LIN {X 0,Y 197.249,Z 148.851,A -85,B 0,C 180,E1 -22908.347,E2 -22908.347} C_VEL
LIN {X 0,Y 203.955,Z 162.722,A -85,B 0,C 180,E1 -22910.636,E2 -22910.636} C_VEL
LIN {X 0,Y 211.585,Z 178.972,A -85,B 0,C 180,E1 -22913.003,E2 -22913.003} C_VEL
LIN {X 0,Y 220.418,Z 193.637,A -85,B 0,C 180,E1 -22915.298,E2 -22915.298} C_VEL
LIN {X 0,Y 228.309,Z 204.661,A -85,B 0,C 180,E1 -22917.116,E2 -22917.116} C_VEL
LIN {X 0,Y 236.225,Z 214.431,A -85,B 0,C 180,E1 -22918.899,E2 -22918.899} C_VEL
LIN {X 0,Y 244.093,Z 223.344,A -85,B 0,C 180,E1 -22920.694,E2 -22920.694} C_VEL
LIN {X 0,Y 253.054,Z 232.486,A -85,B 0,C 180,E1 -22922.712,E2 -22922.712} C_VEL
LIN {X 0,Y 265.026,Z 242.947,A -85,B 0,C 180,E1 -22925.262,E2 -22925.262} C_VEL
LIN {X 0,Y 274.484,Z 250.352,A -85,B 0,C 180,E1 -22927.182,E2 -22927.182} C_VEL
LIN {X 0,Y 288.212,Z 260.222,A -85,B 0,C 180,E1 -22929.853,E2 -22929.853} C_VEL
LIN {X 0,Y 298.287,Z 267.559,A -85,B 0,C 180,E1 -22931.898,E2 -22931.898} C_VEL
LIN {X 0,Y 305.08,Z 272.256,A -85,B 0,C 180,E1 -22933.433,E2 -22933.433} C_VEL
LIN {X 0,Y 312.318,Z 277.42,A -85,B 0,C 180,E1 -22935.376,E2 -22935.376} C_VEL
LIN {X 0,Y 318.689,Z 281.394,A -85,B 0,C 180,E1 -22937.26,E2 -22937.26} C_VEL
LIN {X 0,Y 322.754,Z 284.082,A -85,B 0,C 180,E1 -22938.698,E2 -22938.698} C_VEL
LIN {X 0,Y 327.517,Z 287.382,A -85,B 0,C 180,E1 -22940.778,E2 -22940.778} C_VEL
LIN {X 0,Y 331.199,Z 289.583,A -85,B 0,C 180,E1 -22942.685,E2 -22942.685} C_VEL
LIN {X 0,Y 333.341,Z 290.665,A -85,B 0,C 180,E1 -22943.949,E2 -22943.949} C_VEL
LIN {X 0,Y 335.097,Z 291.438,A -85,B 0,C 180,E1 -22945.188,E2 -22945.188} C_VEL
LIN {X 0,Y 336.519,Z 291.973,A -85,B 0,C 180,E1 -22946.408,E2 -22946.408} C_VEL
LIN {X 0,Y 337.607,Z 292.379,A -85,B 0,C 180,E1 -22947.719,E2 -22947.719} C_VEL
LIN {X 0,Y 338.251,Z 292.675,A -85,B 0,C 180,E1 -22950,E2 -22950} C_VEL
LIN {X 0,Y 338.048,Z 292.601,A -85,B 0,C 180,E1 -22951.191,E2 -22951.191} C_VEL
LIN {X 0,Y 337.513,Z 292.336,A -85,B 0,C 180,E1 -22952.387,E2 -22952.387} C_VEL
LIN {X 0,Y 336.541,Z 291.937,A -85,B 0,C 180,E1 -22953.592,E2 -22953.592} C_VEL
LIN {X 0,Y 335.068,Z 291.43,A -85,B 0,C 180,E1 -22954.813,E2 -22954.813} C_VEL
LIN {X 0,Y 332.494,Z 290.279,A -85,B 0,C 180,E1 -22956.569,E2 -22956.569} C_VEL
LIN {X 0,Y 328.762,Z 288.14,A -85,B 0,C 180,E1 -22958.606,E2 -22958.606} C_VEL
LIN {X 0,Y 324.582,Z 285.413,A -85,B 0,C 180,E1 -22960.528,E2 -22960.528} C_VEL
LIN {X 0,Y 321.255,Z 283.009,A -85,B 0,C 180,E1 -22961.879,E2 -22961.879} C_VEL
LIN {X 0,Y 317.5,Z 280.688,A -85,B 0,C 180,E1 -22963.108,E2 -22963.108} C_VEL
LIN {X 0,Y 312.326,Z 277.399,A -85,B 0,C 180,E1 -22964.63,E2 -22964.63} C_VEL
LIN {X 0,Y 305.085,Z 272.238,A -85,B 0,C 180,E1 -22966.567,E2 -22966.567} C_VEL
LIN {X 0,Y 298.242,Z 267.54,A -85,B 0,C 180,E1 -22968.1,E2 -22968.1} C_VEL
LIN {X 0,Y 288.203,Z 260.253,A -85,B 0,C 180,E1 -22970.142,E2 -22970.142} C_VEL
LIN {X 0,Y 274.482,Z 250.358,A -85,B 0,C 180,E1 -22972.817,E2 -22972.817} C_VEL
LIN {X 0,Y 261.474,Z 240.063,A -85,B 0,C 180,E1 -22975.471,E2 -22975.471} C_VEL
LIN {X 0,Y 249.16,Z 228.707,A -85,B 0,C 180,E1 -22978.153,E2 -22978.153} C_VEL
LIN {X 0,Y 238.844,Z 217.453,A -85,B 0,C 180,E1 -22980.505,E2 -22980.505} C_VEL
LIN {X 0,Y 230.334,Z 207.17,A -85,B 0,C 180,E1 -22982.453,E2 -22982.453} C_VEL
LIN {X 0,Y 221.932,Z 195.931,A -85,B 0,C 180,E1 -22984.341,E2 -22984.341} C_VEL
LIN {X 0,Y 212.893,Z 181.335,A -85,B 0,C 180,E1 -22986.633,E2 -22986.633} C_VEL
LIN {X 0,Y 205.541,Z 166.4,A -85,B 0,C 180,E1 -22988.838,E2 -22988.838} C_VEL
LIN {X 0,Y 199.792,Z 153.911,A -85,B 0,C 180,E1 -22990.767,E2 -22990.767} C_VEL
LIN {X 0,Y 193.529,Z 142.055,A -85,B 0,C 180,E1 -22992.985,E2 -22992.985} C_VEL
LIN {X 0,Y 186.555,Z 130.722,A -85,B 0,C 180,E1 -22995.639,E2 -22995.639} C_VEL
LIN {X 0,Y 180.732,Z 122.331,A -85,B 0,C 180,E1 -22998.061,E2 -22998.061} C_VEL
LIN {X 0,Y 177.666,Z 118.067,A -85,B 0,C 180,E1 -22999.441,E2 -22999.441} C_VEL
LIN {X 0,Y 175.344,Z 114.811,A -85,B 0,C 180,E1 -23000.548,E2 -23000.548} C_VEL
LIN {X 0,Y 174.533,Z 113.689,A -85,B 0,C 180,E1 -23000.947,E2 -23000.947} C_VEL
LIN {X 0,Y 172.411,Z 111.468,A -85,B 0,C 180,E1 -23001.978,E2 -23001.978} C_VEL
LIN {X 0,Y 171.489,Z 109.19,A -85,B 0,C 180,E1 -23002.717,E2 -23002.717} C_VEL
LIN {X 0,Y 171.421,Z 108.64,A -85,B 0,C 180,E1 -23003.526,E2 -23003.526} C_VEL
LIN {X 0,Y 171.454,Z 108.625,A -85,B 0,C 180,E1 -23009.406,E2 -23009.406} C_VEL
LIN {X 0,Y 171.467,Z 108.596,A -85,B 0,C 180,E1 -23014.385,E2 -23014.385} C_VEL
LIN {X 0,Y 171.578,Z 108.565,A -85,B 0,C 180,E1 -23020.873,E2 -23020.873} C_VEL
LIN {X 0,Y 171.611,Z 108.609,A -85,B 0,C 180,E1 -23025.777,E2 -23025.777} C_VEL
LIN {X 0,Y 171.874,Z 108.522,A -85,B 0,C 180,E1 -23030.588,E2 -23030.588} C_VEL
LIN {X 0,Y 171.824,Z 108.582,A -85,B 0,C 180,E1 -23035.309,E2 -23035.309} C_VEL
LIN {X 0,Y 172.332,Z 108.463,A -85,B 0,C 180,E1 -23040.001,E2 -23040.001} C_VEL
LIN {X 0,Y 171.825,Z 108.582,A -85,B 0,C 180,E1 -23044.694,E2 -23044.694} C_VEL
LIN {X 0,Y 171.875,Z 108.52,A -85,B 0,C 180,E1 -23049.415,E2 -23049.415} C_VEL
LIN {X 0,Y 171.612,Z 108.605,A -85,B 0,C 180,E1 -23054.225,E2 -23054.225} C_VEL
LIN {X 0,Y 171.546,Z 108.567,A -85,B 0,C 180,E1 -23059.563,E2 -23059.563} C_VEL
LIN {X 0,Y 171.464,Z 108.592,A -85,B 0,C 180,E1 -23065.612,E2 -23065.612} C_VEL
LIN {X 0,Y 171.458,Z 108.627,A -85,B 0,C 180,E1 -23070.596,E2 -23070.596} C_VEL
LIN {X 0,Y 171.39,Z 108.743,A -85,B 0,C 180,E1 -23076.393,E2 -23076.393} C_VEL
LIN {X 0,Y 171.537,Z 109.44,A -85,B 0,C 180,E1 -23076.997,E2 -23076.997} C_VEL
LIN {X 0,Y 172.996,Z 112.3,A -85,B 0,C 180,E1 -23077.948,E2 -23077.948} C_VEL
LIN {X 0,Y 175.529,Z 115.405,A -85,B 0,C 180,E1 -23079.186,E2 -23079.186} C_VEL
LIN {X 0,Y 178.477,Z 119.92,A -85,B 0,C 180,E1 -23080.599,E2 -23080.599} C_VEL
LIN {X 0,Y 184.499,Z 130.115,A -85,B 0,C 180,E1 -23083.289,E2 -23083.289} C_VEL
LIN {X 0,Y 191.502,Z 143.407,A -85,B 0,C 180,E1 -23086.135,E2 -23086.135} C_VEL
LIN {X 0,Y 197.916,Z 158.306,A -85,B 0,C 180,E1 -23088.591,E2 -23088.591} C_VEL
LIN {X 0,Y 199.96,Z 163.853,A -85,B 0,C 180,E1 -23089.359,E2 -23089.359} C_VEL
LIN {X 0,Y 201.429,Z 175.146,A -85,B 0,C 180,E1 -23090.228,E2 -23090.228} C_VEL
LIN {X 0,Y 199.153,Z 216.376,A -85,B 0,C 180,E1 -23091.646,E2 -23091.646} C_VEL
LIN {X 0,Y 197.784,Z 228.213,A -85,B 0,C 180,E1 -23092.303,E2 -23092.303} C_VEL
LIN {X 0,Y 195.345,Z 241.739,A -85,B 0,C 180,E1 -23093.425,E2 -23093.425} C_VEL
LIN {X 0,Y 192.877,Z 252.257,A -85,B 0,C 180,E1 -23094.659,E2 -23094.659} C_VEL
LIN {X 0,Y 190.358,Z 261.529,A -85,B 0,C 180,E1 -23096.054,E2 -23096.054} C_VEL
LIN {X 0,Y 187.531,Z 270.468,A -85,B 0,C 180,E1 -23097.721,E2 -23097.721} C_VEL
LIN {X 0,Y 184.597,Z 278.993,A -85,B 0,C 180,E1 -23099.705,E2 -23099.705} C_VEL
LIN {X 0,Y 181.871,Z 286.209,A -85,B 0,C 180,E1 -23101.747,E2 -23101.747} C_VEL
LIN {X 0,Y 179.429,Z 292.408,A -85,B 0,C 180,E1 -23103.855,E2 -23103.855} C_VEL
LIN {X 0,Y 176.866,Z 298.948,A -85,B 0,C 180,E1 -23106.587,E2 -23106.587} C_VEL
LIN {X 0,Y 174.91,Z 303.447,A -85,B 0,C 180,E1 -23108.8,E2 -23108.8} C_VEL
LIN {X 0,Y 172.569,Z 308.94,A -85,B 0,C 180,E1 -23112.215,E2 -23112.215} C_VEL
LIN {X 0,Y 170.793,Z 313.267,A -85,B 0,C 180,E1 -23115.706,E2 -23115.706} C_VEL
LIN {X 0,Y 170.011,Z 315.639,A -85,B 0,C 180,E1 -23118.071,E2 -23118.071} C_VEL
LIN {X 0,Y 169.173,Z 318.289,A -85,B 0,C 180,E1 -23121.899,E2 -23121.899} C_VEL
LIN {X 0,Y 168.933,Z 319.901,A -85,B 0,C 180,E1 -23125.227,E2 -23125.227} C_VEL
LIN {X 0,Y 168.87,Z 320.494,A -85,B 0,C 180,E1 -23127.615,E2 -23127.615} C_VEL
LIN {X 0,Y 168.972,Z 320.653,A -85,B 0,C 180,E1 -23130,E2 -23130} C_VEL
LIN {X 0,Y 168.86,Z 320.506,A -85,B 0,C 180,E1 -23132.196,E2 -23132.196} C_VEL
LIN {X 0,Y 168.236,Z 320.196,A -85,B 0,C 180,E1 -23134.188,E2 -23134.188} C_VEL
LIN {X 0,Y 166.772,Z 319.56,A -85,B 0,C 180,E1 -23136.148,E2 -23136.148} C_VEL
LIN {X 0,Y 163.599,Z 317.346,A -85,B 0,C 180,E1 -23140.084,E2 -23140.084} C_VEL
LIN {X 0,Y 163.022,Z 315.76,A -85,B 0,C 180,E1 -23142.09,E2 -23142.09} C_VEL
LIN {X 0,Y 163.126,Z 315.16,A -85,B 0,C 180,E1 -23142.755,E2 -23142.755} C_VEL
LIN {X 0,Y 164.417,Z 311.833,A -85,B 0,C 180,E1 -23146.131,E2 -23146.131} C_VEL
LIN {X 0,Y 166.597,Z 307.089,A -85,B 0,C 180,E1 -23149.724,E2 -23149.724} C_VEL
LIN {X 0,Y 169.325,Z 301.068,A -85,B 0,C 180,E1 -23153.223,E2 -23153.223} C_VEL
LIN {X 0,Y 172.062,Z 294.712,A -85,B 0,C 180,E1 -23156.169,E2 -23156.169} C_VEL
LIN {X 0,Y 174.324,Z 289.27,A -85,B 0,C 180,E1 -23158.275,E2 -23158.275} C_VEL
LIN {X 0,Y 177.778,Z 280.721,A -85,B 0,C 180,E1 -23160.925,E2 -23160.925} C_VEL
LIN {X 0,Y 180.792,Z 272.546,A -85,B 0,C 180,E1 -23162.972,E2 -23162.972} C_VEL
LIN {X 0,Y 183.673,Z 264.04,A -85,B 0,C 180,E1 -23164.692,E2 -23164.692} C_VEL
LIN {X 0,Y 186.227,Z 255.328,A -85,B 0,C 180,E1 -23166.133,E2 -23166.133} C_VEL
LIN {X 0,Y 188.758,Z 245.575,A -85,B 0,C 180,E1 -23167.399,E2 -23167.399} C_VEL
LIN {X 0,Y 190.887,Z 235.498,A -85,B 0,C 180,E1 -23168.411,E2 -23168.411} C_VEL
LIN {X 0,Y 192.569,Z 225.064,A -85,B 0,C 180,E1 -23169.19,E2 -23169.19} C_VEL
LIN {X 0,Y 193.702,Z 215.053,A -85,B 0,C 180,E1 -23169.708,E2 -23169.708} C_VEL
LIN {X 0,Y 195.936,Z 174.885,A -85,B 0,C 180,E1 -23171.126,E2 -23171.126} C_VEL
LIN {X 0,Y 194.533,Z 165.779,A -85,B 0,C 180,E1 -23171.925,E2 -23171.925} C_VEL
LIN {X 0,Y 189.336,Z 152.816,A -85,B 0,C 180,E1 -23174.008,E2 -23174.008} C_VEL
LIN {X 0,Y 184.339,Z 142.18,A -85,B 0,C 180,E1 -23176.098,E2 -23176.098} C_VEL
LIN {X 0,Y 178.821,Z 131.98,A -85,B 0,C 180,E1 -23178.555,E2 -23178.555} C_VEL
LIN {X 0,Y 174.215,Z 124.228,A -85,B 0,C 180,E1 -23180.779,E2 -23180.779} C_VEL
LIN {X 0,Y 171.17,Z 119.458,A -85,B 0,C 180,E1 -23182.355,E2 -23182.355} C_VEL
LIN {X 0,Y 168.703,Z 116.19,A -85,B 0,C 180,E1 -23183.675,E2 -23183.675} C_VEL
LIN {X 0,Y 167.928,Z 114.836,A -85,B 0,C 180,E1 -23184.131,E2 -23184.131} C_VEL
LIN {X 0,Y 165.515,Z 112.604,A -85,B 0,C 180,E1 -23185.46,E2 -23185.46} C_VEL
LIN {X 0,Y 164.436,Z 110.069,A -85,B 0,C 180,E1 -23186.42,E2 -23186.42} C_VEL
LIN {X 0,Y 164.371,Z 109.526,A -85,B 0,C 180,E1 -23187.273,E2 -23187.273} C_VEL
LIN {X 0,Y 164.341,Z 109.475,A -85,B 0,C 180,E1 -23191.938,E2 -23191.938} C_VEL
LIN {X 0,Y 164.412,Z 109.472,A -85,B 0,C 180,E1 -23194.692,E2 -23194.692} C_VEL
LIN {X 0,Y 164.486,Z 109.448,A -85,B 0,C 180,E1 -23200.05,E2 -23200.05} C_VEL
LIN {X 0,Y 164.555,Z 109.481,A -85,B 0,C 180,E1 -23205.151,E2 -23205.151} C_VEL
LIN {X 0,Y 164.799,Z 109.4,A -85,B 0,C 180,E1 -23210.177,E2 -23210.177} C_VEL
LIN {X 0,Y 164.848,Z 109.412,A -85,B 0,C 180,E1 -23212.65,E2 -23212.65} C_VEL
LIN {X 0,Y 165.051,Z 109.389,A -85,B 0,C 180,E1 -23217.558,E2 -23217.558} C_VEL
LIN {X 0,Y 165.294,Z 109.338,A -85,B 0,C 180,E1 -23219.999,E2 -23219.999} C_VEL
LIN {X 0,Y 164.773,Z 109.46,A -85,B 0,C 180,E1 -23224.892,E2 -23224.892} C_VEL
LIN {X 0,Y 164.847,Z 109.415,A -85,B 0,C 180,E1 -23227.347,E2 -23227.347} C_VEL
LIN {X 0,Y 164.75,Z 109.414,A -85,B 0,C 180,E1 -23231.145,E2 -23231.145} C_VEL
LIN {X 0,Y 164.504,Z 109.453,A -85,B 0,C 180,E1 -23237.4,E2 -23237.4} C_VEL
LIN {X 0,Y 164.473,Z 109.452,A -85,B 0,C 180,E1 -23239.988,E2 -23239.988} C_VEL
LIN {X 0,Y 164.391,Z 109.471,A -85,B 0,C 180,E1 -23246.132,E2 -23246.132} C_VEL
LIN {X 0,Y 164.386,Z 109.49,A -85,B 0,C 180,E1 -23252.376,E2 -23252.376} C_VEL
LIN {X 0,Y 164.379,Z 109.808,A -85,B 0,C 180,E1 -23253.765,E2 -23253.765} C_VEL
LIN {X 0,Y 164.762,Z 111.134,A -85,B 0,C 180,E1 -23254.406,E2 -23254.406} C_VEL
LIN {X 0,Y 166.407,Z 113.664,A -85,B 0,C 180,E1 -23255.436,E2 -23255.436} C_VEL
LIN {X 0,Y 168.264,Z 115.23,A -85,B 0,C 180,E1 -23256.431,E2 -23256.431} C_VEL
LIN {X 0,Y 170.431,Z 118.649,A -85,B 0,C 180,E1 -23257.647,E2 -23257.647} C_VEL
LIN {X 0,Y 172.036,Z 120.352,A -85,B 0,C 180,E1 -23258.452,E2 -23258.452} C_VEL
LIN {X 0,Y 174.587,Z 123.964,A -85,B 0,C 180,E1 -23259.73,E2 -23259.73} C_VEL
LIN {X 0,Y 180.798,Z 132.935,A -85,B 0,C 180,E1 -23262.578,E2 -23262.578} C_VEL
LIN {X 0,Y 187.184,Z 143.115,A -85,B 0,C 180,E1 -23265.221,E2 -23265.221} C_VEL
LIN {X 0,Y 192.938,Z 153.571,A -85,B 0,C 180,E1 -23267.425,E2 -23267.425} C_VEL
LIN {X 0,Y 199.185,Z 166.731,A -85,B 0,C 180,E1 -23269.68,E2 -23269.68} C_VEL
LIN {X 0,Y 206.418,Z 182.52,A -85,B 0,C 180,E1 -23272.061,E2 -23272.061} C_VEL
LIN {X 0,Y 215.064,Z 197.26,A -85,B 0,C 180,E1 -23274.444,E2 -23274.444} C_VEL
LIN {X 0,Y 223.339,Z 209.17,A -85,B 0,C 180,E1 -23276.499,E2 -23276.499} C_VEL
LIN {X 0,Y 232.197,Z 220.346,A -85,B 0,C 180,E1 -23278.733,E2 -23278.733} C_VEL
LIN {X 0,Y 242.571,Z 232.02,A -85,B 0,C 180,E1 -23281.341,E2 -23281.341} C_VEL
LIN {X 0,Y 252.676,Z 241.802,A -85,B 0,C 180,E1 -23283.766,E2 -23283.766} C_VEL
LIN {X 0,Y 265.356,Z 252.232,A -85,B 0,C 180,E1 -23286.592,E2 -23286.592} C_VEL
LIN {X 0,Y 278.476,Z 261.599,A -85,B 0,C 180,E1 -23289.309,E2 -23289.309} C_VEL
LIN {X 0,Y 289.053,Z 268.912,A -85,B 0,C 180,E1 -23291.482,E2 -23291.482} C_VEL
LIN {X 0,Y 298.771,Z 275.703,A -85,B 0,C 180,E1 -23293.604,E2 -23293.604} C_VEL
LIN {X 0,Y 305.376,Z 280.454,A -85,B 0,C 180,E1 -23295.336,E2 -23295.336} C_VEL
LIN {X 0,Y 310.985,Z 284.089,A -85,B 0,C 180,E1 -23296.939,E2 -23296.939} C_VEL
LIN {X 0,Y 315.669,Z 286.962,A -85,B 0,C 180,E1 -23298.441,E2 -23298.441} C_VEL
LIN {X 0,Y 320.624,Z 290.479,A -85,B 0,C 180,E1 -23300.531,E2 -23300.531} C_VEL
LIN {X 0,Y 324.649,Z 292.977,A -85,B 0,C 180,E1 -23302.537,E2 -23302.537} C_VEL
LIN {X 0,Y 326.924,Z 294.152,A -85,B 0,C 180,E1 -23303.83,E2 -23303.83} C_VEL
LIN {X 0,Y 328.806,Z 295.053,A -85,B 0,C 180,E1 -23305.095,E2 -23305.095} C_VEL
LIN {X 0,Y 330.806,Z 295.849,A -85,B 0,C 180,E1 -23306.865,E2 -23306.865} C_VEL
LIN {X 0,Y 331.375,Z 296.043,A -85,B 0,C 180,E1 -23307.569,E2 -23307.569} C_VEL
LIN {X 0,Y 331.909,Z 296.335,A -85,B 0,C 180,E1 -23308.787,E2 -23308.787} C_VEL
LIN {X 0,Y 332.2,Z 296.363,A -85,B 0,C 180,E1 -23310,E2 -23310} C_VEL
LIN {X 0,Y 331.968,Z 296.293,A -85,B 0,C 180,E1 -23311.213,E2 -23311.213} C_VEL
LIN {X 0,Y 330.817,Z 295.838,A -85,B 0,C 180,E1 -23313.167,E2 -23313.167} C_VEL
LIN {X 0,Y 328.762,Z 295.057,A -85,B 0,C 180,E1 -23314.905,E2 -23314.905} C_VEL
LIN {X 0,Y 325.647,Z 293.552,A -85,B 0,C 180,E1 -23316.908,E2 -23316.908} C_VEL
LIN {X 0,Y 322.095,Z 291.417,A -85,B 0,C 180,E1 -23318.786,E2 -23318.786} C_VEL
LIN {X 0,Y 319.072,Z 289.452,A -85,B 0,C 180,E1 -23320.149,E2 -23320.149} C_VEL
LIN {X 0,Y 315.63,Z 286.991,A -85,B 0,C 180,E1 -23321.56,E2 -23321.56} C_VEL
LIN {X 0,Y 310.43,Z 283.751,A -85,B 0,C 180,E1 -23323.223,E2 -23323.223} C_VEL
LIN {X 0,Y 305.191,Z 280.327,A -85,B 0,C 180,E1 -23324.722,E2 -23324.722} C_VEL
LIN {X 0,Y 298.731,Z 275.688,A -85,B 0,C 180,E1 -23326.398,E2 -23326.398} C_VEL
LIN {X 0,Y 291.763,Z 270.889,A -85,B 0,C 180,E1 -23327.927,E2 -23327.927} C_VEL
LIN {X 0,Y 283.58,Z 265.098,A -85,B 0,C 180,E1 -23329.654,E2 -23329.654} C_VEL
LIN {X 0,Y 269.952,Z 255.539,A -85,B 0,C 180,E1 -23332.452,E2 -23332.452} C_VEL
LIN {X 0,Y 256.607,Z 245.181,A -85,B 0,C 180,E1 -23335.339,E2 -23335.339} C_VEL
LIN {X 0,Y 244.393,Z 233.939,A -85,B 0,C 180,E1 -23338.204,E2 -23338.204} C_VEL
LIN {X 0,Y 233.764,Z 222.194,A -85,B 0,C 180,E1 -23340.871,E2 -23340.871} C_VEL
LIN {X 0,Y 224.299,Z 210.426,A -85,B 0,C 180,E1 -23343.261,E2 -23343.261} C_VEL
LIN {X 0,Y 216.729,Z 199.81,A -85,B 0,C 180,E1 -23345.139,E2 -23345.139} C_VEL
LIN {X 0,Y 207.695,Z 184.907,A -85,B 0,C 180,E1 -23347.561,E2 -23347.561} C_VEL
LIN {X 0,Y 200.524,Z 169.929,A -85,B 0,C 180,E1 -23349.848,E2 -23349.848} C_VEL
LIN {X 0,Y 195.182,Z 158.13,A -85,B 0,C 180,E1 -23351.748,E2 -23351.748} C_VEL
LIN {X 0,Y 189.114,Z 146.414,A -85,B 0,C 180,E1 -23354.026,E2 -23354.026} C_VEL
LIN {X 0,Y 182.638,Z 135.7,A -85,B 0,C 180,E1 -23356.637,E2 -23356.637} C_VEL
LIN {X 0,Y 177.066,Z 127.573,A -85,B 0,C 180,E1 -23359.088,E2 -23359.088} C_VEL
LIN {X 0,Y 174.22,Z 123.534,A -85,B 0,C 180,E1 -23360.444,E2 -23360.444} C_VEL
LIN {X 0,Y 171.411,Z 119.592,A -85,B 0,C 180,E1 -23361.865,E2 -23361.865} C_VEL
LIN {X 0,Y 169.031,Z 116.717,A -85,B 0,C 180,E1 -23363.111,E2 -23363.111} C_VEL
LIN {X 0,Y 167.918,Z 114.799,A -85,B 0,C 180,E1 -23363.761,E2 -23363.761} C_VEL
LIN {X 0,Y 165.692,Z 112.821,A -85,B 0,C 180,E1 -23364.979,E2 -23364.979} C_VEL
LIN {X 0,Y 164.418,Z 110.047,A -85,B 0,C 180,E1 -23366.035,E2 -23366.035} C_VEL
LIN {X 0,Y 164.346,Z 109.51,A -85,B 0,C 180,E1 -23366.924,E2 -23366.924} C_VEL
LIN {X 0,Y 164.402,Z 109.507,A -85,B 0,C 180,E1 -23369.139,E2 -23369.139} C_VEL
LIN {X 0,Y 164.415,Z 109.476,A -85,B 0,C 180,E1 -23374.695,E2 -23374.695} C_VEL
LIN {X 0,Y 164.484,Z 109.45,A -85,B 0,C 180,E1 -23380.052,E2 -23380.052} C_VEL
LIN {X 0,Y 164.554,Z 109.487,A -85,B 0,C 180,E1 -23385.153,E2 -23385.153} C_VEL
LIN {X 0,Y 164.798,Z 109.402,A -85,B 0,C 180,E1 -23390.18,E2 -23390.18} C_VEL
LIN {X 0,Y 164.847,Z 109.415,A -85,B 0,C 180,E1 -23392.653,E2 -23392.653} C_VEL
LIN {X 0,Y 165.05,Z 109.386,A -85,B 0,C 180,E1 -23397.561,E2 -23397.561} C_VEL
LIN {X 0,Y 165.294,Z 109.338,A -85,B 0,C 180,E1 -23400.001,E2 -23400.001} C_VEL
LIN {X 0,Y 164.775,Z 109.461,A -85,B 0,C 180,E1 -23404.895,E2 -23404.895} C_VEL
LIN {X 0,Y 164.848,Z 109.412,A -85,B 0,C 180,E1 -23407.35,E2 -23407.35} C_VEL
LIN {X 0,Y 164.752,Z 109.413,A -85,B 0,C 180,E1 -23411.148,E2 -23411.148} C_VEL
LIN {X 0,Y 164.506,Z 109.447,A -85,B 0,C 180,E1 -23417.402,E2 -23417.402} C_VEL
LIN {X 0,Y 164.475,Z 109.45,A -85,B 0,C 180,E1 -23419.99,E2 -23419.99} C_VEL
LIN {X 0,Y 164.39,Z 109.468,A -85,B 0,C 180,E1 -23426.131,E2 -23426.131} C_VEL
LIN {X 0,Y 164.387,Z 109.5,A -85,B 0,C 180,E1 -23432.379,E2 -23432.379} C_VEL
LIN {X 0,Y 164.405,Z 109.859,A -85,B 0,C 180,E1 -23433.413,E2 -23433.413} C_VEL
LIN {X 0,Y 164.724,Z 111.046,A -85,B 0,C 180,E1 -23433.999,E2 -23433.999} C_VEL
LIN {X 0,Y 166.276,Z 113.495,A -85,B 0,C 180,E1 -23434.981,E2 -23434.981} C_VEL
LIN {X 0,Y 168.272,Z 115.282,A -85,B 0,C 180,E1 -23436.062,E2 -23436.062} C_VEL
LIN {X 0,Y 170.321,Z 118.538,A -85,B 0,C 180,E1 -23437.213,E2 -23437.213} C_VEL
LIN {X 0,Y 172.25,Z 121.065,A -85,B 0,C 180,E1 -23438.211,E2 -23438.211} C_VEL
LIN {X 0,Y 176.093,Z 127.356,A -85,B 0,C 180,E1 -23440.152,E2 -23440.152} C_VEL
LIN {X 0,Y 180.443,Z 134.78,A -85,B 0,C 180,E1 -23442.184,E2 -23442.184} C_VEL
LIN {X 0,Y 187.165,Z 147.789,A -85,B 0,C 180,E1 -23445.086,E2 -23445.086} C_VEL
LIN {X 0,Y 193.156,Z 162.188,A -85,B 0,C 180,E1 -23447.533,E2 -23447.533} C_VEL
LIN {X 0,Y 194.789,Z 166.664,A -85,B 0,C 180,E1 -23448.185,E2 -23448.185} C_VEL
LIN {X 0,Y 195.994,Z 175.498,A -85,B 0,C 180,E1 -23448.918,E2 -23448.918} C_VEL
LIN {X 0,Y 193.644,Z 216.029,A -85,B 0,C 180,E1 -23450.334,E2 -23450.334} C_VEL
LIN {X 0,Y 192.225,Z 227.822,A -85,B 0,C 180,E1 -23450.992,E2 -23450.992} C_VEL
LIN {X 0,Y 189.688,Z 241.549,A -85,B 0,C 180,E1 -23452.147,E2 -23452.147} C_VEL
LIN {X 0,Y 187.127,Z 252.066,A -85,B 0,C 180,E1 -23453.4,E2 -23453.4} C_VEL
LIN {X 0,Y 184.516,Z 261.338,A -85,B 0,C 180,E1 -23454.824,E2 -23454.824} C_VEL
LIN {X 0,Y 181.577,Z 270.278,A -85,B 0,C 180,E1 -23456.527,E2 -23456.527} C_VEL
LIN {X 0,Y 178.477,Z 278.802,A -85,B 0,C 180,E1 -23458.55,E2 -23458.55} C_VEL
LIN {X 0,Y 175.628,Z 286.017,A -85,B 0,C 180,E1 -23460.646,E2 -23460.646} C_VEL
LIN {X 0,Y 173.06,Z 292.217,A -85,B 0,C 180,E1 -23462.815,E2 -23462.815} C_VEL
LIN {X 0,Y 170.338,Z 298.757,A -85,B 0,C 180,E1 -23465.632,E2 -23465.632} C_VEL
LIN {X 0,Y 168.283,Z 303.256,A -85,B 0,C 180,E1 -23467.922,E2 -23467.922} C_VEL
LIN {X 0,Y 165.811,Z 308.749,A -85,B 0,C 180,E1 -23471.465,E2 -23471.465} C_VEL
LIN {X 0,Y 163.872,Z 313.075,A -85,B 0,C 180,E1 -23475.089,E2 -23475.089} C_VEL
LIN {X 0,Y 163.038,Z 315.447,A -85,B 0,C 180,E1 -23477.553,E2 -23477.553} C_VEL
LIN {X 0,Y 162.398,Z 317.251,A -85,B 0,C 180,E1 -23480.032,E2 -23480.032} C_VEL
LIN {X 0,Y 161.851,Z 319.71,A -85,B 0,C 180,E1 -23485.018,E2 -23485.018} C_VEL
LIN {X 0,Y 161.8,Z 320.304,A -85,B 0,C 180,E1 -23487.511,E2 -23487.511} C_VEL
LIN {X 0,Y 161.884,Z 320.463,A -85,B 0,C 180,E1 -23490,E2 -23490} C_VEL
LIN {X 0,Y 161.763,Z 320.303,A -85,B 0,C 180,E1 -23492.49,E2 -23492.49} C_VEL
LIN {X 0,Y 161.794,Z 319.708,A -85,B 0,C 180,E1 -23494.984,E2 -23494.984} C_VEL
LIN {X 0,Y 162.398,Z 317.251,A -85,B 0,C 180,E1 -23499.968,E2 -23499.968} C_VEL
LIN {X 0,Y 163.126,Z 315.16,A -85,B 0,C 180,E1 -23502.755,E2 -23502.755} C_VEL
LIN {X 0,Y 163.143,Z 313.326,A -85,B 0,C 180,E1 -23504.719,E2 -23504.719} C_VEL
LIN {X 0,Y 161.821,Z 309.895,A -85,B 0,C 180,E1 -23507.961,E2 -23507.961} C_VEL
LIN {X 0,Y 160.964,Z 305.907,A -85,B 0,C 180,E1 -23511.171,E2 -23511.171} C_VEL
LIN {X 0,Y 161.707,Z 303.078,A -85,B 0,C 180,E1 -23513.017,E2 -23513.017} C_VEL
LIN {X 0,Y 164.978,Z 296.213,A -85,B 0,C 180,E1 -23516.542,E2 -23516.542} C_VEL
LIN {X 0,Y 168.08,Z 289.079,A -85,B 0,C 180,E1 -23519.427,E2 -23519.427} C_VEL
LIN {X 0,Y 171.72,Z 280.531,A -85,B 0,C 180,E1 -23522.144,E2 -23522.144} C_VEL
LIN {X 0,Y 174.87,Z 272.356,A -85,B 0,C 180,E1 -23524.24,E2 -23524.24} C_VEL
LIN {X 0,Y 177.852,Z 263.849,A -85,B 0,C 180,E1 -23526.001,E2 -23526.001} C_VEL
LIN {X 0,Y 180.527,Z 255.137,A -85,B 0,C 180,E1 -23527.466,E2 -23527.466} C_VEL
LIN {X 0,Y 183.166,Z 245.385,A -85,B 0,C 180,E1 -23528.748,E2 -23528.748} C_VEL
LIN {X 0,Y 185.377,Z 235.307,A -85,B 0,C 180,E1 -23529.774,E2 -23529.774} C_VEL
LIN {X 0,Y 187.117,Z 224.921,A -85,B 0,C 180,E1 -23530.56,E2 -23530.56} C_VEL
LIN {X 0,Y 188.213,Z 215.719,A -85,B 0,C 180,E1 -23531.053,E2 -23531.053} C_VEL
LIN {X 0,Y 190.577,Z 176.151,A -85,B 0,C 180,E1 -23532.475,E2 -23532.475} C_VEL
LIN {X 0,Y 189.414,Z 168.518,A -85,B 0,C 180,E1 -23533.182,E2 -23533.182} C_VEL
LIN {X 0,Y 184.374,Z 155.859,A -85,B 0,C 180,E1 -23535.341,E2 -23535.341} C_VEL
LIN {X 0,Y 180.064,Z 146.476,A -85,B 0,C 180,E1 -23537.273,E2 -23537.273} C_VEL
LIN {X 0,Y 173.97,Z 134.873,A -85,B 0,C 180,E1 -23540.203,E2 -23540.203} C_VEL
LIN {X 0,Y 170.38,Z 128.995,A -85,B 0,C 180,E1 -23542.056,E2 -23542.056} C_VEL
LIN {X 0,Y 167.958,Z 125.065,A -85,B 0,C 180,E1 -23543.395,E2 -23543.395} C_VEL
LIN {X 0,Y 165.346,Z 121.319,A -85,B 0,C 180,E1 -23544.898,E2 -23544.898} C_VEL
LIN {X 0,Y 162.352,Z 117.927,A -85,B 0,C 180,E1 -23546.685,E2 -23546.685} C_VEL
LIN {X 0,Y 161.131,Z 115.819,A -85,B 0,C 180,E1 -23547.517,E2 -23547.517} C_VEL
LIN {X 0,Y 158.699,Z 113.734,A -85,B 0,C 180,E1 -23549.091,E2 -23549.091} C_VEL
LIN {X 0,Y 157.378,Z 110.942,A -85,B 0,C 180,E1 -23550.394,E2 -23550.394} C_VEL
LIN {X 0,Y 157.297,Z 110.404,A -85,B 0,C 180,E1 -23551.294,E2 -23551.294} C_VEL
LIN {X 0,Y 157.312,Z 110.379,A -85,B 0,C 180,E1 -23556.29,E2 -23556.29} C_VEL
LIN {X 0,Y 157.425,Z 110.324,A -85,B 0,C 180,E1 -23561.788,E2 -23561.788} C_VEL
LIN {X 0,Y 157.555,Z 110.332,A -85,B 0,C 180,E1 -23567.111,E2 -23567.111} C_VEL
LIN {X 0,Y 157.728,Z 110.281,A -85,B 0,C 180,E1 -23569.732,E2 -23569.732} C_VEL
LIN {X 0,Y 157.805,Z 110.283,A -85,B 0,C 180,E1 -23572.321,E2 -23572.321} C_VEL
LIN {X 0,Y 158.257,Z 110.214,A -85,B 0,C 180,E1 -23579.999,E2 -23579.999} C_VEL
LIN {X 0,Y 157.804,Z 110.286,A -85,B 0,C 180,E1 -23587.677,E2 -23587.677} C_VEL
LIN {X 0,Y 157.68,Z 110.295,A -85,B 0,C 180,E1 -23591.315,E2 -23591.315} C_VEL
LIN {X 0,Y 157.478,Z 110.355,A -85,B 0,C 180,E1 -23595.53,E2 -23595.53} C_VEL
LIN {X 0,Y 157.369,Z 110.344,A -85,B 0,C 180,E1 -23600.931,E2 -23600.931} C_VEL
LIN {X 0,Y 157.312,Z 110.35,A -85,B 0,C 180,E1 -23606.682,E2 -23606.682} C_VEL
LIN {X 0,Y 157.327,Z 110.672,A -85,B 0,C 180,E1 -23609.706,E2 -23609.706} C_VEL
LIN {X 0,Y 157.673,Z 111.834,A -85,B 0,C 180,E1 -23610.464,E2 -23610.464} C_VEL
LIN {X 0,Y 159.295,Z 114.459,A -85,B 0,C 180,E1 -23611.702,E2 -23611.702} C_VEL
LIN {X 0,Y 161.541,Z 116.336,A -85,B 0,C 180,E1 -23613.129,E2 -23613.129} C_VEL
LIN {X 0,Y 163.725,Z 119.727,A -85,B 0,C 180,E1 -23614.549,E2 -23614.549} C_VEL
LIN {X 0,Y 165.506,Z 121.571,A -85,B 0,C 180,E1 -23615.576,E2 -23615.576} C_VEL
LIN {X 0,Y 168.074,Z 125.13,A -85,B 0,C 180,E1 -23617.04,E2 -23617.04} C_VEL
LIN {X 0,Y 170.065,Z 127.966,A -85,B 0,C 180,E1 -23618.117,E2 -23618.117} C_VEL
LIN {X 0,Y 173.015,Z 132.118,A -85,B 0,C 180,E1 -23619.62,E2 -23619.62} C_VEL
LIN {X 0,Y 179.466,Z 141.769,A -85,B 0,C 180,E1 -23622.626,E2 -23622.626} C_VEL
LIN {X 0,Y 186.55,Z 154.082,A -85,B 0,C 180,E1 -23625.61,E2 -23625.61} C_VEL
LIN {X 0,Y 193.357,Z 168.202,A -85,B 0,C 180,E1 -23628.259,E2 -23628.259} C_VEL
LIN {X 0,Y 201.66,Z 186.76,A -85,B 0,C 180,E1 -23631.183,E2 -23631.183} C_VEL
LIN {X 0,Y 210.82,Z 202.552,A -85,B 0,C 180,E1 -23633.837,E2 -23633.837} C_VEL
LIN {X 0,Y 218.416,Z 213.86,A -85,B 0,C 180,E1 -23635.949,E2 -23635.949} C_VEL
LIN {X 0,Y 226.087,Z 223.874,A -85,B 0,C 180,E1 -23638.099,E2 -23638.099} C_VEL
LIN {X 0,Y 234.396,Z 233.608,A -85,B 0,C 180,E1 -23640.401,E2 -23640.401} C_VEL
LIN {X 0,Y 242.744,Z 242.295,A -85,B 0,C 180,E1 -23642.631,E2 -23642.631} C_VEL
LIN {X 0,Y 252.117,Z 250.547,A -85,B 0,C 180,E1 -23644.953,E2 -23644.953} C_VEL
LIN {X 0,Y 263.452,Z 259.254,A -85,B 0,C 180,E1 -23647.567,E2 -23647.567} C_VEL
LIN {X 0,Y 276.16,Z 267.978,A -85,B 0,C 180,E1 -23650.322,E2 -23650.322} C_VEL
LIN {X 0,Y 284.361,Z 273.416,A -85,B 0,C 180,E1 -23652.085,E2 -23652.085} C_VEL
LIN {X 0,Y 292.562,Z 278.981,A -85,B 0,C 180,E1 -23653.92,E2 -23653.92} C_VEL
LIN {X 0,Y 299.5,Z 283.906,A -85,B 0,C 180,E1 -23655.701,E2 -23655.701} C_VEL
LIN {X 0,Y 304.721,Z 287.346,A -85,B 0,C 180,E1 -23657.18,E2 -23657.18} C_VEL
LIN {X 0,Y 309.791,Z 290.459,A -85,B 0,C 180,E1 -23658.786,E2 -23658.786} C_VEL
LIN {X 0,Y 315.026,Z 294.121,A -85,B 0,C 180,E1 -23661.016,E2 -23661.016} C_VEL
LIN {X 0,Y 318.718,Z 296.426,A -85,B 0,C 180,E1 -23662.873,E2 -23662.873} C_VEL
LIN {X 0,Y 322.183,Z 298.125,A -85,B 0,C 180,E1 -23664.994,E2 -23664.994} C_VEL
LIN {X 0,Y 323.932,Z 298.879,A -85,B 0,C 180,E1 -23666.373,E2 -23666.373} C_VEL
LIN {X 0,Y 324.99,Z 299.282,A -85,B 0,C 180,E1 -23667.521,E2 -23667.521} C_VEL
LIN {X 0,Y 325.6,Z 299.576,A -85,B 0,C 180,E1 -23668.763,E2 -23668.763} C_VEL
LIN {X 0,Y 325.887,Z 299.626,A -85,B 0,C 180,E1 -23670,E2 -23670} C_VEL
LIN {X 0,Y 325.644,Z 299.548,A -85,B 0,C 180,E1 -23671.237,E2 -23671.237} C_VEL
LIN {X 0,Y 325.003,Z 299.267,A -85,B 0,C 180,E1 -23672.479,E2 -23672.479} C_VEL
LIN {X 0,Y 323.812,Z 298.812,A -85,B 0,C 180,E1 -23673.733,E2 -23673.733} C_VEL
LIN {X 0,Y 322.137,Z 298.141,A -85,B 0,C 180,E1 -23675.006,E2 -23675.006} C_VEL
LIN {X 0,Y 318.717,Z 296.398,A -85,B 0,C 180,E1 -23677.126,E2 -23677.126} C_VEL
LIN {X 0,Y 315.014,Z 294.154,A -85,B 0,C 180,E1 -23678.985,E2 -23678.985} C_VEL
LIN {X 0,Y 311.792,Z 291.962,A -85,B 0,C 180,E1 -23680.389,E2 -23680.389} C_VEL
LIN {X 0,Y 307.827,Z 289.27,A -85,B 0,C 180,E1 -23681.858,E2 -23681.858} C_VEL
LIN {X 0,Y 302.572,Z 285.977,A -85,B 0,C 180,E1 -23683.431,E2 -23683.431} C_VEL
LIN {X 0,Y 296.455,Z 281.723,A -85,B 0,C 180,E1 -23685.116,E2 -23685.116} C_VEL
LIN {X 0,Y 289.818,Z 277.125,A -85,B 0,C 180,E1 -23686.697,E2 -23686.697} C_VEL
LIN {X 0,Y 278.762,Z 269.658,A -85,B 0,C 180,E1 -23689.132,E2 -23689.132} C_VEL
LIN {X 0,Y 265.34,Z 260.556,A -85,B 0,C 180,E1 -23692.025,E2 -23692.025} C_VEL
LIN {X 0,Y 252.111,Z 250.57,A -85,B 0,C 180,E1 -23695.043,E2 -23695.043} C_VEL
LIN {X 0,Y 241.108,Z 240.677,A -85,B 0,C 180,E1 -23697.8,E2 -23697.8} C_VEL
LIN {X 0,Y 230.663,Z 229.419,A -85,B 0,C 180,E1 -23700.625,E2 -23700.625} C_VEL
LIN {X 0,Y 221.648,Z 218.141,A -85,B 0,C 180,E1 -23703.147,E2 -23703.147} C_VEL
LIN {X 0,Y 214.413,Z 208.09,A -85,B 0,C 180,E1 -23705.177,E2 -23705.177} C_VEL
LIN {X 0,Y 205.964,Z 194.581,A -85,B 0,C 180,E1 -23707.516,E2 -23707.516} C_VEL
LIN {X 0,Y 198.391,Z 179.951,A -85,B 0,C 180,E1 -23709.901,E2 -23709.901} C_VEL
LIN {X 0,Y 191.023,Z 163.165,A -85,B 0,C 180,E1 -23712.625,E2 -23712.625} C_VEL
LIN {X 0,Y 185.207,Z 151.603,A -85,B 0,C 180,E1 -23714.934,E2 -23714.934} C_VEL
LIN {X 0,Y 178.857,Z 140.821,A -85,B 0,C 180,E1 -23717.643,E2 -23717.643} C_VEL
LIN {X 0,Y 173.664,Z 133.023,A -85,B 0,C 180,E1 -23720.063,E2 -23720.063} C_VEL
LIN {X 0,Y 170.302,Z 128.315,A -85,B 0,C 180,E1 -23721.757,E2 -23721.757} C_VEL
LIN {X 0,Y 168.072,Z 125.15,A -85,B 0,C 180,E1 -23722.96,E2 -23722.96} C_VEL
LIN {X 0,Y 165.507,Z 121.559,A -85,B 0,C 180,E1 -23724.424,E2 -23724.424} C_VEL
LIN {X 0,Y 162.242,Z 117.704,A -85,B 0,C 180,E1 -23726.383,E2 -23726.383} C_VEL
LIN {X 0,Y 161.118,Z 115.823,A -85,B 0,C 180,E1 -23727.146,E2 -23727.146} C_VEL
LIN {X 0,Y 158.711,Z 113.744,A -85,B 0,C 180,E1 -23728.705,E2 -23728.705} C_VEL
LIN {X 0,Y 157.448,Z 111.13,A -85,B 0,C 180,E1 -23729.858,E2 -23729.858} C_VEL
LIN {X 0,Y 157.281,Z 110.434,A -85,B 0,C 180,E1 -23730.928,E2 -23730.928} C_VEL
LIN {X 0,Y 157.319,Z 110.349,A -85,B 0,C 180,E1 -23733.467,E2 -23733.467} C_VEL
LIN {X 0,Y 157.393,Z 110.335,A -85,B 0,C 180,E1 -23739.669,E2 -23739.669} C_VEL
LIN {X 0,Y 157.478,Z 110.355,A -85,B 0,C 180,E1 -23744.47,E2 -23744.47} C_VEL
LIN {X 0,Y 157.726,Z 110.283,A -85,B 0,C 180,E1 -23749.735,E2 -23749.735} C_VEL
LIN {X 0,Y 157.804,Z 110.286,A -85,B 0,C 180,E1 -23752.323,E2 -23752.323} C_VEL
LIN {X 0,Y 158.257,Z 110.214,A -85,B 0,C 180,E1 -23760.001,E2 -23760.001} C_VEL
LIN {X 0,Y 157.805,Z 110.283,A -85,B 0,C 180,E1 -23767.679,E2 -23767.679} C_VEL
LIN {X 0,Y 157.682,Z 110.294,A -85,B 0,C 180,E1 -23771.318,E2 -23771.318} C_VEL
LIN {X 0,Y 157.48,Z 110.347,A -85,B 0,C 180,E1 -23775.533,E2 -23775.533} C_VEL
LIN {X 0,Y 157.371,Z 110.343,A -85,B 0,C 180,E1 -23780.934,E2 -23780.934} C_VEL
LIN {X 0,Y 157.311,Z 110.347,A -85,B 0,C 180,E1 -23786.682,E2 -23786.682} C_VEL
LIN {X 0,Y 157.338,Z 110.664,A -85,B 0,C 180,E1 -23789.339,E2 -23789.339} C_VEL
LIN {X 0,Y 157.676,Z 111.894,A -85,B 0,C 180,E1 -23790.097,E2 -23790.097} C_VEL
LIN {X 0,Y 159.428,Z 114.585,A -85,B 0,C 180,E1 -23791.412,E2 -23791.412} C_VEL
LIN {X 0,Y 161.45,Z 116.178,A -85,B 0,C 180,E1 -23792.689,E2 -23792.689} C_VEL
LIN {X 0,Y 163.426,Z 119.387,A -85,B 0,C 180,E1 -23793.992,E2 -23793.992} C_VEL
LIN {X 0,Y 165.465,Z 121.563,A -85,B 0,C 180,E1 -23795.178,E2 -23795.178} C_VEL
LIN {X 0,Y 168.996,Z 126.628,A -85,B 0,C 180,E1 -23797.18,E2 -23797.18} C_VEL
LIN {X 0,Y 173.112,Z 133.543,A -85,B 0,C 180,E1 -23799.373,E2 -23799.373} C_VEL
LIN {X 0,Y 177.249,Z 141.057,A -85,B 0,C 180,E1 -23801.416,E2 -23801.416} C_VEL
LIN {X 0,Y 182.975,Z 152.42,A -85,B 0,C 180,E1 -23804.027,E2 -23804.027} C_VEL
LIN {X 0,Y 188.898,Z 167.151,A -85,B 0,C 180,E1 -23806.602,E2 -23806.602} C_VEL
LIN {X 0,Y 189.902,Z 170.694,A -85,B 0,C 180,E1 -23807.064,E2 -23807.064} C_VEL
LIN {X 0,Y 190.633,Z 176.75,A -85,B 0,C 180,E1 -23807.57,E2 -23807.57} C_VEL
LIN {X 0,Y 188.228,Z 215.844,A -85,B 0,C 180,E1 -23808.953,E2 -23808.953} C_VEL
LIN {X 0,Y 186.791,Z 227.498,A -85,B 0,C 180,E1 -23809.615,E2 -23809.615} C_VEL
LIN {X 0,Y 184.134,Z 241.358,A -85,B 0,C 180,E1 -23810.791,E2 -23810.791} C_VEL
LIN {X 0,Y 181.471,Z 251.875,A -85,B 0,C 180,E1 -23812.062,E2 -23812.062} C_VEL
LIN {X 0,Y 178.768,Z 261.148,A -85,B 0,C 180,E1 -23813.515,E2 -23813.515} C_VEL
LIN {X 0,Y 175.702,Z 270.088,A -85,B 0,C 180,E1 -23815.25,E2 -23815.25} C_VEL
LIN {X 0,Y 172.426,Z 278.611,A -85,B 0,C 180,E1 -23817.312,E2 -23817.312} C_VEL
LIN {X 0,Y 169.464,Z 285.827,A -85,B 0,C 180,E1 -23819.467,E2 -23819.467} C_VEL
LIN {X 0,Y 166.744,Z 292.026,A -85,B 0,C 180,E1 -23821.695,E2 -23821.695} C_VEL
LIN {X 0,Y 163.867,Z 298.565,A -85,B 0,C 180,E1 -23824.603,E2 -23824.603} C_VEL
LIN {X 0,Y 161.709,Z 303.065,A -85,B 0,C 180,E1 -23826.974,E2 -23826.974} C_VEL
LIN {X 0,Y 159.058,Z 308.557,A -85,B 0,C 180,E1 -23830.647,E2 -23830.647} C_VEL
LIN {X 0,Y 156.977,Z 312.883,A -85,B 0,C 180,E1 -23834.418,E2 -23834.418} C_VEL
LIN {X 0,Y 156.064,Z 315.256,A -85,B 0,C 180,E1 -23836.988,E2 -23836.988} C_VEL
LIN {X 0,Y 155.398,Z 317.06,A -85,B 0,C 180,E1 -23839.578,E2 -23839.578} C_VEL
LIN {X 0,Y 154.754,Z 319.519,A -85,B 0,C 180,E1 -23844.789,E2 -23844.789} C_VEL
LIN {X 0,Y 154.715,Z 320.234,A -85,B 0,C 180,E1 -23847.983,E2 -23847.983} C_VEL
LIN {X 0,Y 154.687,Z 320.264,A -85,B 0,C 180,E1 -23851.695,E2 -23851.695} C_VEL
LIN {X 0,Y 154.714,Z 319.518,A -85,B 0,C 180,E1 -23855.213,E2 -23855.213} C_VEL
LIN {X 0,Y 155.398,Z 317.06,A -85,B 0,C 180,E1 -23860.422,E2 -23860.422} C_VEL
LIN {X 0,Y 156.498,Z 314.103,A -85,B 0,C 180,E1 -23864.3,E2 -23864.3} C_VEL
LIN {X 0,Y 158.276,Z 310.111,A -85,B 0,C 180,E1 -23868.109,E2 -23868.109} C_VEL
LIN {X 0,Y 160.765,Z 304.981,A -85,B 0,C 180,E1 -23871.813,E2 -23871.813} C_VEL
LIN {X 0,Y 161.707,Z 303.078,A -85,B 0,C 180,E1 -23873.017,E2 -23873.017} C_VEL
LIN {X 0,Y 162.542,Z 300.132,A -85,B 0,C 180,E1 -23874.803,E2 -23874.803} C_VEL
LIN {X 0,Y 162.373,Z 294.788,A -85,B 0,C 180,E1 -23877.751,E2 -23877.751} C_VEL
LIN {X 0,Y 162.479,Z 288.906,A -85,B 0,C 180,E1 -23880.553,E2 -23880.553} C_VEL
LIN {X 0,Y 163.709,Z 284.917,A -85,B 0,C 180,E1 -23882.048,E2 -23882.048} C_VEL
LIN {X 0,Y 168.188,Z 274.433,A -85,B 0,C 180,E1 -23885.069,E2 -23885.069} C_VEL
LIN {X 0,Y 171.73,Z 265.01,A -85,B 0,C 180,E1 -23887.131,E2 -23887.131} C_VEL
LIN {X 0,Y 174.949,Z 254.947,A -85,B 0,C 180,E1 -23888.879,E2 -23888.879} C_VEL
LIN {X 0,Y 177.686,Z 245.194,A -85,B 0,C 180,E1 -23890.181,E2 -23890.181} C_VEL
LIN {X 0,Y 179.974,Z 235.117,A -85,B 0,C 180,E1 -23891.221,E2 -23891.221} C_VEL
LIN {X 0,Y 181.769,Z 224.844,A -85,B 0,C 180,E1 -23892.007,E2 -23892.007} C_VEL
LIN {X 0,Y 182.929,Z 215.535,A -85,B 0,C 180,E1 -23892.51,E2 -23892.51} C_VEL
LIN {X 0,Y 185.331,Z 177.404,A -85,B 0,C 180,E1 -23893.902,E2 -23893.902} C_VEL
LIN {X 0,Y 184.432,Z 171.348,A -85,B 0,C 180,E1 -23894.492,E2 -23894.492} C_VEL
LIN {X 0,Y 178.803,Z 157.055,A -85,B 0,C 180,E1 -23897.097,E2 -23897.097} C_VEL
LIN {X 0,Y 173.972,Z 146.985,A -85,B 0,C 180,E1 -23899.446,E2 -23899.446} C_VEL
LIN {X 0,Y 169.459,Z 138.488,A -85,B 0,C 180,E1 -23901.815,E2 -23901.815} C_VEL
LIN {X 0,Y 166.762,Z 133.86,A -85,B 0,C 180,E1 -23903.325,E2 -23903.325} C_VEL
LIN {X 0,Y 164.68,Z 130.506,A -85,B 0,C 180,E1 -23904.547,E2 -23904.547} C_VEL
LIN {X 0,Y 161.836,Z 126.539,A -85,B 0,C 180,E1 -23906.285,E2 -23906.285} C_VEL
LIN {X 0,Y 159.195,Z 123.116,A -85,B 0,C 180,E1 -23908.009,E2 -23908.009} C_VEL
LIN {X 0,Y 158.433,Z 121.997,A -85,B 0,C 180,E1 -23908.544,E2 -23908.544} C_VEL
LIN {X 0,Y 155.958,Z 119.433,A -85,B 0,C 180,E1 -23910.283,E2 -23910.283} C_VEL
LIN {X 0,Y 154.508,Z 116.921,A -85,B 0,C 180,E1 -23911.469,E2 -23911.469} C_VEL
LIN {X 0,Y 151.873,Z 114.912,A -85,B 0,C 180,E1 -23913.546,E2 -23913.546} C_VEL
LIN {X 0,Y 150.42,Z 112.222,A -85,B 0,C 180,E1 -23915.066,E2 -23915.066} C_VEL
LIN {X 0,Y 150.273,Z 111.344,A -85,B 0,C 180,E1 -23916.209,E2 -23916.209} C_VEL
LIN {X 0,Y 150.368,Z 111.201,A -85,B 0,C 180,E1 -23920.901,E2 -23920.901} C_VEL
LIN {X 0,Y 150.462,Z 111.225,A -85,B 0,C 180,E1 -23926.493,E2 -23926.493} C_VEL
LIN {X 0,Y 150.654,Z 111.163,A -85,B 0,C 180,E1 -23929.244,E2 -23929.244} C_VEL
LIN {X 0,Y 150.741,Z 111.158,A -85,B 0,C 180,E1 -23931.958,E2 -23931.958} C_VEL
LIN {X 0,Y 151.218,Z 111.09,A -85,B 0,C 180,E1 -23939.999,E2 -23939.999} C_VEL
LIN {X 0,Y 150.74,Z 111.161,A -85,B 0,C 180,E1 -23948.039,E2 -23948.039} C_VEL
LIN {X 0,Y 150.611,Z 111.176,A -85,B 0,C 180,E1 -23951.5,E2 -23951.5} C_VEL
LIN {X 0,Y 150.382,Z 111.224,A -85,B 0,C 180,E1 -23956.283,E2 -23956.283} C_VEL
LIN {X 0,Y 150.35,Z 111.216,A -85,B 0,C 180,E1 -23960.791,E2 -23960.791} C_VEL
LIN {X 0,Y 150.273,Z 111.484,A -85,B 0,C 180,E1 -23964.614,E2 -23964.614} C_VEL
LIN {X 0,Y 150.537,Z 112.6,A -85,B 0,C 180,E1 -23965.506,E2 -23965.506} C_VEL
LIN {X 0,Y 152.166,Z 115.239,A -85,B 0,C 180,E1 -23967.084,E2 -23967.084} C_VEL
LIN {X 0,Y 154.873,Z 117.366,A -85,B 0,C 180,E1 -23969.196,E2 -23969.196} C_VEL
LIN {X 0,Y 156.746,Z 120.483,A -85,B 0,C 180,E1 -23970.684,E2 -23970.684} C_VEL
LIN {X 0,Y 159.003,Z 122.704,A -85,B 0,C 180,E1 -23972.224,E2 -23972.224} C_VEL
LIN {X 0,Y 161.604,Z 126.336,A -85,B 0,C 180,E1 -23973.955,E2 -23973.955} C_VEL
LIN {X 0,Y 162.843,Z 127.862,A -85,B 0,C 180,E1 -23974.717,E2 -23974.717} C_VEL
LIN {X 0,Y 166.743,Z 133.333,A -85,B 0,C 180,E1 -23977.007,E2 -23977.007} C_VEL
LIN {X 0,Y 171.617,Z 140.439,A -85,B 0,C 180,E1 -23979.59,E2 -23979.59} C_VEL
LIN {X 0,Y 177.843,Z 150.485,A -85,B 0,C 180,E1 -23982.565,E2 -23982.565} C_VEL
LIN {X 0,Y 183.604,Z 161.163,A -85,B 0,C 180,E1 -23985.082,E2 -23985.082} C_VEL
LIN {X 0,Y 189.329,Z 173.723,A -85,B 0,C 180,E1 -23987.435,E2 -23987.435} C_VEL
LIN {X 0,Y 197.41,Z 191.903,A -85,B 0,C 180,E1 -23990.415,E2 -23990.415} C_VEL
LIN {X 0,Y 205.534,Z 206.267,A -85,B 0,C 180,E1 -23992.958,E2 -23992.958} C_VEL
LIN {X 0,Y 211.649,Z 215.879,A -85,B 0,C 180,E1 -23994.853,E2 -23994.853} C_VEL
LIN {X 0,Y 219.324,Z 226.579,A -85,B 0,C 180,E1 -23997.26,E2 -23997.26} C_VEL
LIN {X 0,Y 227.672,Z 236.684,A -85,B 0,C 180,E1 -23999.804,E2 -23999.804} C_VEL
LIN {X 0,Y 237.403,Z 246.978,A -85,B 0,C 180,E1 -24002.635,E2 -24002.635} C_VEL
LIN {X 0,Y 249.267,Z 257.136,A -85,B 0,C 180,E1 -24005.741,E2 -24005.741} C_VEL
LIN {X 0,Y 260.653,Z 265.424,A -85,B 0,C 180,E1 -24008.467,E2 -24008.467} C_VEL
LIN {X 0,Y 274.189,Z 274.177,A -85,B 0,C 180,E1 -24011.508,E2 -24011.508} C_VEL
LIN {X 0,Y 286.558,Z 282.141,A -85,B 0,C 180,E1 -24014.349,E2 -24014.349} C_VEL
LIN {X 0,Y 293.526,Z 286.959,A -85,B 0,C 180,E1 -24016.147,E2 -24016.147} C_VEL
LIN {X 0,Y 299.38,Z 290.826,A -85,B 0,C 180,E1 -24017.803,E2 -24017.803} C_VEL
LIN {X 0,Y 304.118,Z 293.788,A -85,B 0,C 180,E1 -24019.346,E2 -24019.346} C_VEL
LIN {X 0,Y 307.593,Z 296.24,A -85,B 0,C 180,E1 -24020.797,E2 -24020.797} C_VEL
LIN {X 0,Y 311.688,Z 298.862,A -85,B 0,C 180,E1 -24022.795,E2 -24022.795} C_VEL
LIN {X 0,Y 315.268,Z 300.736,A -85,B 0,C 180,E1 -24024.884,E2 -24024.884} C_VEL
LIN {X 0,Y 317.02,Z 301.483,A -85,B 0,C 180,E1 -24026.187,E2 -24026.187} C_VEL
LIN {X 0,Y 318.338,Z 301.983,A -85,B 0,C 180,E1 -24027.469,E2 -24027.469} C_VEL
LIN {X 0,Y 319.043,Z 302.306,A -85,B 0,C 180,E1 -24028.738,E2 -24028.738} C_VEL
LIN {X 0,Y 319.34,Z 302.389,A -85,B 0,C 180,E1 -24030,E2 -24030} C_VEL
LIN {X 0,Y 319.076,Z 302.291,A -85,B 0,C 180,E1 -24031.262,E2 -24031.262} C_VEL
LIN {X 0,Y 318.35,Z 301.976,A -85,B 0,C 180,E1 -24032.531,E2 -24032.531} C_VEL
LIN {X 0,Y 316.969,Z 301.476,A -85,B 0,C 180,E1 -24033.846,E2 -24033.846} C_VEL
LIN {X 0,Y 315.244,Z 300.746,A -85,B 0,C 180,E1 -24035.116,E2 -24035.116} C_VEL
LIN {X 0,Y 311.688,Z 298.848,A -85,B 0,C 180,E1 -24037.204,E2 -24037.204} C_VEL
LIN {X 0,Y 307.571,Z 296.228,A -85,B 0,C 180,E1 -24039.204,E2 -24039.204} C_VEL
LIN {X 0,Y 304.076,Z 293.785,A -85,B 0,C 180,E1 -24040.655,E2 -24040.655} C_VEL
LIN {X 0,Y 298.2,Z 290.114,A -85,B 0,C 180,E1 -24042.544,E2 -24042.544} C_VEL
LIN {X 0,Y 290.562,Z 284.868,A -85,B 0,C 180,E1 -24044.65,E2 -24044.65} C_VEL
LIN {X 0,Y 282.364,Z 279.518,A -85,B 0,C 180,E1 -24046.616,E2 -24046.616} C_VEL
LIN {X 0,Y 271.45,Z 272.509,A -85,B 0,C 180,E1 -24049.093,E2 -24049.093} C_VEL
LIN {X 0,Y 257.968,Z 263.62,A -85,B 0,C 180,E1 -24052.14,E2 -24052.14} C_VEL
LIN {X 0,Y 244.943,Z 253.698,A -85,B 0,C 180,E1 -24055.341,E2 -24055.341} C_VEL
LIN {X 0,Y 234.937,Z 244.533,A -85,B 0,C 180,E1 -24058.06,E2 -24058.06} C_VEL
LIN {X 0,Y 226.019,Z 234.789,A -85,B 0,C 180,E1 -24060.692,E2 -24060.692} C_VEL
LIN {X 0,Y 217.554,Z 224.13,A -85,B 0,C 180,E1 -24063.311,E2 -24063.311} C_VEL
LIN {X 0,Y 209.754,Z 212.978,A -85,B 0,C 180,E1 -24065.762,E2 -24065.762} C_VEL
LIN {X 0,Y 202.385,Z 200.877,A -85,B 0,C 180,E1 -24068.024,E2 -24068.024} C_VEL
LIN {X 0,Y 195.361,Z 187.636,A -85,B 0,C 180,E1 -24070.289,E2 -24070.289} C_VEL
LIN {X 0,Y 186.413,Z 167.126,A -85,B 0,C 180,E1 -24073.744,E2 -24073.744} C_VEL
LIN {X 0,Y 180.886,Z 155.904,A -85,B 0,C 180,E1 -24076.083,E2 -24076.083} C_VEL
LIN {X 0,Y 175.116,Z 145.952,A -85,B 0,C 180,E1 -24078.699,E2 -24078.699} C_VEL
LIN {X 0,Y 169.22,Z 136.861,A -85,B 0,C 180,E1 -24081.649,E2 -24081.649} C_VEL
LIN {X 0,Y 164.999,Z 130.833,A -85,B 0,C 180,E1 -24083.992,E2 -24083.992} C_VEL
LIN {X 0,Y 161.939,Z 126.651,A -85,B 0,C 180,E1 -24085.844,E2 -24085.844} C_VEL
LIN {X 0,Y 159.299,Z 123.257,A -85,B 0,C 180,E1 -24087.56,E2 -24087.56} C_VEL
LIN {X 0,Y 158.403,Z 121.97,A -85,B 0,C 180,E1 -24088.187,E2 -24088.187} C_VEL
LIN {X 0,Y 155.932,Z 119.406,A -85,B 0,C 180,E1 -24089.925,E2 -24089.925} C_VEL
LIN {X 0,Y 154.494,Z 116.951,A -85,B 0,C 180,E1 -24091.098,E2 -24091.098} C_VEL
LIN {X 0,Y 151.768,Z 114.786,A -85,B 0,C 180,E1 -24093.261,E2 -24093.261} C_VEL
LIN {X 0,Y 150.331,Z 111.844,A -85,B 0,C 180,E1 -24094.987,E2 -24094.987} C_VEL
LIN {X 0,Y 150.28,Z 111.28,A -85,B 0,C 180,E1 -24096.579,E2 -24096.579} C_VEL
LIN {X 0,Y 150.366,Z 111.204,A -85,B 0,C 180,E1 -24100.904,E2 -24100.904} C_VEL
LIN {X 0,Y 150.46,Z 111.225,A -85,B 0,C 180,E1 -24106.495,E2 -24106.495} C_VEL
LIN {X 0,Y 150.653,Z 111.165,A -85,B 0,C 180,E1 -24109.247,E2 -24109.247} C_VEL
LIN {X 0,Y 150.74,Z 111.161,A -85,B 0,C 180,E1 -24111.961,E2 -24111.961} C_VEL
LIN {X 0,Y 151.218,Z 111.09,A -85,B 0,C 180,E1 -24120.001,E2 -24120.001} C_VEL
LIN {X 0,Y 150.741,Z 111.158,A -85,B 0,C 180,E1 -24128.042,E2 -24128.042} C_VEL
LIN {X 0,Y 150.612,Z 111.175,A -85,B 0,C 180,E1 -24131.503,E2 -24131.503} C_VEL
LIN {X 0,Y 150.384,Z 111.217,A -85,B 0,C 180,E1 -24136.286,E2 -24136.286} C_VEL
LIN {X 0,Y 150.352,Z 111.214,A -85,B 0,C 180,E1 -24140.793,E2 -24140.793} C_VEL
LIN {X 0,Y 150.304,Z 111.566,A -85,B 0,C 180,E1 -24144.336,E2 -24144.336} C_VEL
LIN {X 0,Y 150.618,Z 112.828,A -85,B 0,C 180,E1 -24145.229,E2 -24145.229} C_VEL
LIN {X 0,Y 152.328,Z 115.408,A -85,B 0,C 180,E1 -24146.844,E2 -24146.844} C_VEL
LIN {X 0,Y 154.79,Z 117.243,A -85,B 0,C 180,E1 -24148.752,E2 -24148.752} C_VEL
LIN {X 0,Y 156.697,Z 120.415,A -85,B 0,C 180,E1 -24150.271,E2 -24150.271} C_VEL
LIN {X 0,Y 158.919,Z 122.589,A -85,B 0,C 180,E1 -24151.789,E2 -24151.789} C_VEL
LIN {X 0,Y 161.394,Z 126.087,A -85,B 0,C 180,E1 -24153.446,E2 -24153.446} C_VEL
LIN {X 0,Y 162.917,Z 128.013,A -85,B 0,C 180,E1 -24154.389,E2 -24154.389} C_VEL
LIN {X 0,Y 165.76,Z 132.096,A -85,B 0,C 180,E1 -24156.084,E2 -24156.084} C_VEL
LIN {X 0,Y 170.849,Z 140.868,A -85,B 0,C 180,E1 -24158.925,E2 -24158.925} C_VEL
LIN {X 0,Y 177.668,Z 154.461,A -85,B 0,C 180,E1 -24162.359,E2 -24162.359} C_VEL
LIN {X 0,Y 182.911,Z 167.231,A -85,B 0,C 180,E1 -24164.818,E2 -24164.818} C_VEL
LIN {X 0,Y 184.854,Z 173.227,A -85,B 0,C 180,E1 -24165.735,E2 -24165.735} C_VEL
LIN {X 0,Y 185.304,Z 178.561,A -85,B 0,C 180,E1 -24166.15,E2 -24166.15} C_VEL
LIN {X 0,Y 182.934,Z 215.658,A -85,B 0,C 180,E1 -24167.492,E2 -24167.492} C_VEL
LIN {X 0,Y 181.384,Z 227.723,A -85,B 0,C 180,E1 -24168.191,E2 -24168.191} C_VEL
LIN {X 0,Y 178.698,Z 241.168,A -85,B 0,C 180,E1 -24169.354,E2 -24169.354} C_VEL
LIN {X 0,Y 175.935,Z 251.685,A -85,B 0,C 180,E1 -24170.643,E2 -24170.643} C_VEL
LIN {X 0,Y 173.112,Z 260.958,A -85,B 0,C 180,E1 -24172.118,E2 -24172.118} C_VEL
LIN {X 0,Y 169.918,Z 269.897,A -85,B 0,C 180,E1 -24173.886,E2 -24173.886} C_VEL
LIN {X 0,Y 166.477,Z 278.419,A -85,B 0,C 180,E1 -24175.988,E2 -24175.988} C_VEL
LIN {X 0,Y 163.362,Z 285.635,A -85,B 0,C 180,E1 -24178.197,E2 -24178.197} C_VEL
LIN {X 0,Y 160.491,Z 291.834,A -85,B 0,C 180,E1 -24180.486,E2 -24180.486} C_VEL
LIN {X 0,Y 157.438,Z 298.373,A -85,B 0,C 180,E1 -24183.487,E2 -24183.487} C_VEL
LIN {X 0,Y 155.191,Z 302.874,A -85,B 0,C 180,E1 -24185.947,E2 -24185.947} C_VEL
LIN {X 0,Y 152.35,Z 308.366,A -85,B 0,C 180,E1 -24189.758,E2 -24189.758} C_VEL
LIN {X 0,Y 150.111,Z 312.691,A -85,B 0,C 180,E1 -24193.685,E2 -24193.685} C_VEL
LIN {X 0,Y 149.118,Z 315.064,A -85,B 0,C 180,E1 -24196.37,E2 -24196.37} C_VEL
LIN {X 0,Y 148.384,Z 316.869,A -85,B 0,C 180,E1 -24199.079,E2 -24199.079} C_VEL
LIN {X 0,Y 147.686,Z 319.328,A -85,B 0,C 180,E1 -24204.539,E2 -24204.539} C_VEL
LIN {X 0,Y 147.628,Z 320.079,A -85,B 0,C 180,E1 -24208.731,E2 -24208.731} C_VEL
LIN {X 0,Y 147.572,Z 319.922,A -85,B 0,C 180,E1 -24212.73,E2 -24212.73} C_VEL
LIN {X 0,Y 147.637,Z 319.327,A -85,B 0,C 180,E1 -24215.463,E2 -24215.463} C_VEL
LIN {X 0,Y 148.384,Z 316.869,A -85,B 0,C 180,E1 -24220.921,E2 -24220.921} C_VEL
LIN {X 0,Y 149.6,Z 313.912,A -85,B 0,C 180,E1 -24224.974,E2 -24224.974} C_VEL
LIN {X 0,Y 151.533,Z 309.92,A -85,B 0,C 180,E1 -24228.945,E2 -24228.945} C_VEL
LIN {X 0,Y 154.153,Z 304.789,A -85,B 0,C 180,E1 -24232.8,E2 -24232.8} C_VEL
LIN {X 0,Y 156.903,Z 299.53,A -85,B 0,C 180,E1 -24235.895,E2 -24235.895} C_VEL
LIN {X 0,Y 159.087,Z 294.943,A -85,B 0,C 180,E1 -24238.168,E2 -24238.168} C_VEL
LIN {X 0,Y 161.901,Z 288.888,A -85,B 0,C 180,E1 -24240.668,E2 -24240.668} C_VEL
LIN {X 0,Y 163.709,Z 284.917,A -85,B 0,C 180,E1 -24242.048,E2 -24242.048} C_VEL
LIN {X 0,Y 164.978,Z 280.84,A -85,B 0,C 180,E1 -24243.479,E2 -24243.479} C_VEL
LIN {X 0,Y 165.417,Z 273.855,A -85,B 0,C 180,E1 -24245.931,E2 -24245.931} C_VEL
LIN {X 0,Y 165.962,Z 266.454,A -85,B 0,C 180,E1 -24248.188,E2 -24248.188} C_VEL
LIN {X 0,Y 167.264,Z 261.528,A -85,B 0,C 180,E1 -24249.238,E2 -24249.238} C_VEL
LIN {X 0,Y 170.526,Z 251.495,A -85,B 0,C 180,E1 -24250.864,E2 -24250.864} C_VEL
LIN {X 0,Y 173.929,Z 238.787,A -85,B 0,C 180,E1 -24252.399,E2 -24252.399} C_VEL
LIN {X 0,Y 176.333,Z 226.185,A -85,B 0,C 180,E1 -24253.446,E2 -24253.446} C_VEL
LIN {X 0,Y 177.689,Z 216.096,A -85,B 0,C 180,E1 -24254.023,E2 -24254.023} C_VEL
LIN {X 0,Y 179.676,Z 187.814,A -85,B 0,C 180,E1 -24255.074,E2 -24255.074} C_VEL
LIN {X 0,Y 180.215,Z 178.567,A -85,B 0,C 180,E1 -24255.414,E2 -24255.414} C_VEL
LIN {X 0,Y 179.44,Z 173.911,A -85,B 0,C 180,E1 -24255.925,E2 -24255.925} C_VEL
LIN {X 0,Y 174.123,Z 160.168,A -85,B 0,C 180,E1 -24258.579,E2 -24258.579} C_VEL
LIN {X 0,Y 168.623,Z 148.626,A -85,B 0,C 180,E1 -24261.494,E2 -24261.494} C_VEL
LIN {X 0,Y 164.055,Z 140.145,A -85,B 0,C 180,E1 -24264.144,E2 -24264.144} C_VEL
LIN {X 0,Y 161.499,Z 135.937,A -85,B 0,C 180,E1 -24265.733,E2 -24265.733} C_VEL
LIN {X 0,Y 158.866,Z 132.252,A -85,B 0,C 180,E1 -24267.443,E2 -24267.443} C_VEL
LIN {X 0,Y 155.878,Z 128.151,A -85,B 0,C 180,E1 -24269.553,E2 -24269.553} C_VEL
LIN {X 0,Y 153.192,Z 124.964,A -85,B 0,C 180,E1 -24271.599,E2 -24271.599} C_VEL
LIN {X 0,Y 152.155,Z 123.296,A -85,B 0,C 180,E1 -24272.489,E2 -24272.489} C_VEL
LIN {X 0,Y 149.554,Z 120.899,A -85,B 0,C 180,E1 -24274.712,E2 -24274.712} C_VEL
LIN {X 0,Y 147.796,Z 117.95,A -85,B 0,C 180,E1 -24276.53,E2 -24276.53} C_VEL
LIN {X 0,Y 145.285,Z 116.18,A -85,B 0,C 180,E1 -24279.14,E2 -24279.14} C_VEL
LIN {X 0,Y 143.695,Z 113.645,A -85,B 0,C 180,E1 -24281.277,E2 -24281.277} C_VEL
LIN {X 0,Y 143.352,Z 112.466,A -85,B 0,C 180,E1 -24282.524,E2 -24282.524} C_VEL
LIN {X 0,Y 143.38,Z 112.12,A -85,B 0,C 180,E1 -24285.812,E2 -24285.812} C_VEL
LIN {X 0,Y 143.596,Z 112.045,A -85,B 0,C 180,E1 -24288.709,E2 -24288.709} C_VEL
LIN {X 0,Y 143.661,Z 112.035,A -85,B 0,C 180,E1 -24291.559,E2 -24291.559} C_VEL
LIN {X 0,Y 144.177,Z 111.966,A -85,B 0,C 180,E1 -24299.998,E2 -24299.998} C_VEL
LIN {X 0,Y 143.66,Z 112.038,A -85,B 0,C 180,E1 -24308.438,E2 -24308.438} C_VEL
LIN {X 0,Y 143.548,Z 112.056,A -85,B 0,C 180,E1 -24311.711,E2 -24311.711} C_VEL
LIN {X 0,Y 143.344,Z 112.373,A -85,B 0,C 180,E1 -24317.658,E2 -24317.658} C_VEL
LIN {X 0,Y 143.644,Z 113.489,A -85,B 0,C 180,E1 -24319.004,E2 -24319.004} C_VEL
LIN {X 0,Y 145.167,Z 116.108,A -85,B 0,C 180,E1 -24321.106,E2 -24321.106} C_VEL
LIN {X 0,Y 147.789,Z 117.939,A -85,B 0,C 180,E1 -24323.84,E2 -24323.84} C_VEL
LIN {X 0,Y 148.541,Z 119.218,A -85,B 0,C 180,E1 -24324.641,E2 -24324.641} C_VEL
LIN {X 0,Y 150.674,Z 122.196,A -85,B 0,C 180,E1 -24326.681,E2 -24326.681} C_VEL
LIN {X 0,Y 152.605,Z 123.816,A -85,B 0,C 180,E1 -24328.259,E2 -24328.259} C_VEL
LIN {X 0,Y 154.706,Z 127.014,A -85,B 0,C 180,E1 -24329.979,E2 -24329.979} C_VEL
LIN {X 0,Y 156.466,Z 128.882,A -85,B 0,C 180,E1 -24331.25,E2 -24331.25} C_VEL
LIN {X 0,Y 159.371,Z 132.801,A -85,B 0,C 180,E1 -24333.261,E2 -24333.261} C_VEL
LIN {X 0,Y 163.876,Z 139.296,A -85,B 0,C 180,E1 -24336.085,E2 -24336.085} C_VEL
LIN {X 0,Y 169.862,Z 148.387,A -85,B 0,C 180,E1 -24339.387,E2 -24339.387} C_VEL
LIN {X 0,Y 175.439,Z 158.051,A -85,B 0,C 180,E1 -24342.153,E2 -24342.153} C_VEL
LIN {X 0,Y 180.411,Z 167.827,A -85,B 0,C 180,E1 -24344.429,E2 -24344.429} C_VEL
LIN {X 0,Y 185.359,Z 179.228,A -85,B 0,C 180,E1 -24346.579,E2 -24346.579} C_VEL
LIN {X 0,Y 193.005,Z 196.634,A -85,B 0,C 180,E1 -24349.546,E2 -24349.546} C_VEL
LIN {X 0,Y 200.895,Z 210.955,A -85,B 0,C 180,E1 -24352.222,E2 -24352.222} C_VEL
LIN {X 0,Y 207.269,Z 221.341,A -85,B 0,C 180,E1 -24354.465,E2 -24354.465} C_VEL
LIN {X 0,Y 214.392,Z 231.546,A -85,B 0,C 180,E1 -24356.962,E2 -24356.962} C_VEL
LIN {X 0,Y 223.291,Z 242.411,A -85,B 0,C 180,E1 -24359.942,E2 -24359.942} C_VEL
LIN {X 0,Y 232.831,Z 252.343,A -85,B 0,C 180,E1 -24362.93,E2 -24362.93} C_VEL
LIN {X 0,Y 242.839,Z 260.806,A -85,B 0,C 180,E1 -24365.733,E2 -24365.733} C_VEL
LIN {X 0,Y 255.896,Z 270.079,A -85,B 0,C 180,E1 -24369.03,E2 -24369.03} C_VEL
LIN {X 0,Y 269.435,Z 278.421,A -85,B 0,C 180,E1 -24372.184,E2 -24372.184} C_VEL
LIN {X 0,Y 280.393,Z 285.104,A -85,B 0,C 180,E1 -24374.792,E2 -24374.792} C_VEL
LIN {X 0,Y 285.854,Z 288.585,A -85,B 0,C 180,E1 -24376.196,E2 -24376.196} C_VEL
LIN {X 0,Y 291.595,Z 292.375,A -85,B 0,C 180,E1 -24377.801,E2 -24377.801} C_VEL
LIN {X 0,Y 297.996,Z 296.411,A -85,B 0,C 180,E1 -24379.813,E2 -24379.813} C_VEL
LIN {X 0,Y 302.938,Z 299.844,A -85,B 0,C 180,E1 -24381.999,E2 -24381.999} C_VEL
LIN {X 0,Y 305.761,Z 301.525,A -85,B 0,C 180,E1 -24383.401,E2 -24383.401} C_VEL
LIN {X 0,Y 308.072,Z 302.749,A -85,B 0,C 180,E1 -24384.764,E2 -24384.764} C_VEL
LIN {X 0,Y 310.034,Z 303.647,A -85,B 0,C 180,E1 -24386.101,E2 -24386.101} C_VEL
LIN {X 0,Y 311.445,Z 304.21,A -85,B 0,C 180,E1 -24387.413,E2 -24387.413} C_VEL
LIN {X 0,Y 312.268,Z 304.541,A -85,B 0,C 180,E1 -24388.71,E2 -24388.71} C_VEL
LIN {X 0,Y 312.597,Z 304.635,A -85,B 0,C 180,E1 -24390,E2 -24390} C_VEL
LIN {X 0,Y 312.295,Z 304.535,A -85,B 0,C 180,E1 -24391.29,E2 -24391.29} C_VEL
LIN {X 0,Y 311.456,Z 304.21,A -85,B 0,C 180,E1 -24392.587,E2 -24392.587} C_VEL
LIN {X 0,Y 309.957,Z 303.644,A -85,B 0,C 180,E1 -24393.933,E2 -24393.933} C_VEL
LIN {X 0,Y 308.059,Z 302.771,A -85,B 0,C 180,E1 -24395.236,E2 -24395.236} C_VEL
LIN {X 0,Y 304.598,Z 300.866,A -85,B 0,C 180,E1 -24397.196,E2 -24397.196} C_VEL
LIN {X 0,Y 299.74,Z 297.634,A -85,B 0,C 180,E1 -24399.447,E2 -24399.447} C_VEL
LIN {X 0,Y 297.937,Z 296.418,A -85,B 0,C 180,E1 -24400.19,E2 -24400.19} C_VEL
LIN {X 0,Y 291.593,Z 292.38,A -85,B 0,C 180,E1 -24402.197,E2 -24402.197} C_VEL
LIN {X 0,Y 283.128,Z 286.834,A -85,B 0,C 180,E1 -24404.518,E2 -24404.518} C_VEL
LIN {X 0,Y 272.155,Z 280.15,A -85,B 0,C 180,E1 -24407.166,E2 -24407.166} C_VEL
LIN {X 0,Y 258.577,Z 271.772,A -85,B 0,C 180,E1 -24410.337,E2 -24410.337} C_VEL
LIN {X 0,Y 245.393,Z 262.792,A -85,B 0,C 180,E1 -24413.587,E2 -24413.587} C_VEL
LIN {X 0,Y 235.297,Z 254.54,A -85,B 0,C 180,E1 -24416.358,E2 -24416.358} C_VEL
LIN {X 0,Y 226.827,Z 246.284,A -85,B 0,C 180,E1 -24418.92,E2 -24418.92} C_VEL
LIN {X 0,Y 218.638,Z 236.898,A -85,B 0,C 180,E1 -24421.591,E2 -24421.591} C_VEL
LIN {X 0,Y 211.785,Z 227.861,A -85,B 0,C 180,E1 -24423.943,E2 -24423.943} C_VEL
LIN {X 0,Y 205.114,Z 218.071,A -85,B 0,C 180,E1 -24426.269,E2 -24426.269} C_VEL
LIN {X 0,Y 198.444,Z 206.703,A -85,B 0,C 180,E1 -24428.617,E2 -24428.617} C_VEL
LIN {X 0,Y 191.23,Z 192.904,A -85,B 0,C 180,E1 -24431.095,E2 -24431.095} C_VEL
LIN {X 0,Y 181.675,Z 170.615,A -85,B 0,C 180,E1 -24435.01,E2 -24435.01} C_VEL
LIN {X 0,Y 176.562,Z 160.043,A -85,B 0,C 180,E1 -24437.326,E2 -24437.326} C_VEL
LIN {X 0,Y 170.998,Z 150.343,A -85,B 0,C 180,E1 -24440.023,E2 -24440.023} C_VEL
LIN {X 0,Y 165.039,Z 140.906,A -85,B 0,C 180,E1 -24443.246,E2 -24443.246} C_VEL
LIN {X 0,Y 161.523,Z 135.96,A -85,B 0,C 180,E1 -24445.341,E2 -24445.341} C_VEL
LIN {X 0,Y 159.046,Z 132.471,A -85,B 0,C 180,E1 -24446.946,E2 -24446.946} C_VEL
LIN {X 0,Y 155.806,Z 128.098,A -85,B 0,C 180,E1 -24449.225,E2 -24449.225} C_VEL
LIN {X 0,Y 153.208,Z 124.989,A -85,B 0,C 180,E1 -24451.208,E2 -24451.208} C_VEL
LIN {X 0,Y 152.335,Z 123.452,A -85,B 0,C 180,E1 -24451.967,E2 -24451.967} C_VEL
LIN {X 0,Y 149.688,Z 121.103,A -85,B 0,C 180,E1 -24454.205,E2 -24454.205} C_VEL
LIN {X 0,Y 147.787,Z 117.956,A -85,B 0,C 180,E1 -24456.16,E2 -24456.16} C_VEL
LIN {X 0,Y 145.167,Z 116.108,A -85,B 0,C 180,E1 -24458.894,E2 -24458.894} C_VEL
LIN {X 0,Y 143.646,Z 113.472,A -85,B 0,C 180,E1 -24460.996,E2 -24460.996} C_VEL
LIN {X 0,Y 143.338,Z 112.387,A -85,B 0,C 180,E1 -24462.341,E2 -24462.341} C_VEL
LIN {X 0,Y 143.594,Z 112.047,A -85,B 0,C 180,E1 -24468.712,E2 -24468.712} C_VEL
LIN {X 0,Y 143.66,Z 112.038,A -85,B 0,C 180,E1 -24471.562,E2 -24471.562} C_VEL
LIN {X 0,Y 144.177,Z 111.966,A -85,B 0,C 180,E1 -24480.002,E2 -24480.002} C_VEL
LIN {X 0,Y 143.661,Z 112.035,A -85,B 0,C 180,E1 -24488.441,E2 -24488.441} C_VEL
LIN {X 0,Y 143.549,Z 112.055,A -85,B 0,C 180,E1 -24491.714,E2 -24491.714} C_VEL
LIN {X 0,Y 143.351,Z 112.404,A -85,B 0,C 180,E1 -24497.384,E2 -24497.384} C_VEL
LIN {X 0,Y 143.642,Z 113.542,A -85,B 0,C 180,E1 -24498.638,E2 -24498.638} C_VEL
LIN {X 0,Y 145.285,Z 116.18,A -85,B 0,C 180,E1 -24500.86,E2 -24500.86} C_VEL
LIN {X 0,Y 148.111,Z 118.306,A -85,B 0,C 180,E1 -24503.788,E2 -24503.788} C_VEL
LIN {X 0,Y 149.91,Z 121.374,A -85,B 0,C 180,E1 -24505.623,E2 -24505.623} C_VEL
LIN {X 0,Y 152.606,Z 123.878,A -85,B 0,C 180,E1 -24507.889,E2 -24507.889} C_VEL
LIN {X 0,Y 154.908,Z 127.231,A -85,B 0,C 180,E1 -24509.752,E2 -24509.752} C_VEL
LIN {X 0,Y 156.482,Z 128.941,A -85,B 0,C 180,E1 -24510.887,E2 -24510.887} C_VEL
LIN {X 0,Y 159.43,Z 132.852,A -85,B 0,C 180,E1 -24512.92,E2 -24512.92} C_VEL
LIN {X 0,Y 162.797,Z 137.975,A -85,B 0,C 180,E1 -24515.081,E2 -24515.081} C_VEL
LIN {X 0,Y 167.258,Z 145.904,A -85,B 0,C 180,E1 -24517.733,E2 -24517.733} C_VEL
LIN {X 0,Y 173.345,Z 158.373,A -85,B 0,C 180,E1 -24521.02,E2 -24521.02} C_VEL
LIN {X 0,Y 177.877,Z 169.702,A -85,B 0,C 180,E1 -24523.315,E2 -24523.315} C_VEL
LIN {X 0,Y 179.892,Z 175.476,A -85,B 0,C 180,E1 -24524.31,E2 -24524.31} C_VEL
LIN {X 0,Y 180.215,Z 178.565,A -85,B 0,C 180,E1 -24524.586,E2 -24524.586} C_VEL
LIN {X 0,Y 177.794,Z 215.057,A -85,B 0,C 180,E1 -24525.922,E2 -24525.922} C_VEL
LIN {X 0,Y 176.347,Z 226.191,A -85,B 0,C 180,E1 -24526.559,E2 -24526.559} C_VEL
LIN {X 0,Y 173.929,Z 238.787,A -85,B 0,C 180,E1 -24527.601,E2 -24527.601} C_VEL
LIN {X 0,Y 170.511,Z 251.495,A -85,B 0,C 180,E1 -24529.132,E2 -24529.132} C_VEL
LIN {X 0,Y 167.567,Z 260.767,A -85,B 0,C 180,E1 -24530.627,E2 -24530.627} C_VEL
LIN {X 0,Y 164.225,Z 269.706,A -85,B 0,C 180,E1 -24532.423,E2 -24532.423} C_VEL
LIN {X 0,Y 160.635,Z 278.229,A -85,B 0,C 180,E1 -24534.57,E2 -24534.57} C_VEL
LIN {X 0,Y 157.355,Z 285.444,A -85,B 0,C 180,E1 -24536.83,E2 -24536.83} C_VEL
LIN {X 0,Y 154.329,Z 291.643,A -85,B 0,C 180,E1 -24539.182,E2 -24539.182} C_VEL
LIN {X 0,Y 151.061,Z 298.181,A -85,B 0,C 180,E1 -24542.274,E2 -24542.274} C_VEL
LIN {X 0,Y 148.732,Z 302.684,A -85,B 0,C 180,E1 -24544.832,E2 -24544.832} C_VEL
LIN {X 0,Y 145.684,Z 308.175,A -85,B 0,C 180,E1 -24548.789,E2 -24548.789} C_VEL
LIN {X 0,Y 143.272,Z 312.5,A -85,B 0,C 180,E1 -24552.883,E2 -24552.883} C_VEL
LIN {X 0,Y 142.202,Z 314.873,A -85,B 0,C 180,E1 -24555.693,E2 -24555.693} C_VEL
LIN {X 0,Y 141.394,Z 316.678,A -85,B 0,C 180,E1 -24558.532,E2 -24558.532} C_VEL
LIN {X 0,Y 140.616,Z 319.138,A -85,B 0,C 180,E1 -24564.263,E2 -24564.263} C_VEL
LIN {X 0,Y 140.572,Z 319.89,A -85,B 0,C 180,E1 -24569.356,E2 -24569.356} C_VEL
LIN {X 0,Y 140.49,Z 319.732,A -85,B 0,C 180,E1 -24572.867,E2 -24572.867} C_VEL
LIN {X 0,Y 140.557,Z 319.136,A -85,B 0,C 180,E1 -24575.739,E2 -24575.739} C_VEL
LIN {X 0,Y 141.394,Z 316.678,A -85,B 0,C 180,E1 -24581.468,E2 -24581.468} C_VEL
LIN {X 0,Y 142.705,Z 313.72,A -85,B 0,C 180,E1 -24585.716,E2 -24585.716} C_VEL
LIN {X 0,Y 144.799,Z 309.728,A -85,B 0,C 180,E1 -24589.862,E2 -24589.862} C_VEL
LIN {X 0,Y 147.603,Z 304.598,A -85,B 0,C 180,E1 -24593.873,E2 -24593.873} C_VEL
LIN {X 0,Y 150.519,Z 299.339,A -85,B 0,C 180,E1 -24597.081,E2 -24597.081} C_VEL
LIN {X 0,Y 153.659,Z 293.02,A -85,B 0,C 180,E1 -24600.206,E2 -24600.206} C_VEL
LIN {X 0,Y 156.582,Z 287.07,A -85,B 0,C 180,E1 -24602.589,E2 -24602.589} C_VEL
LIN {X 0,Y 159.833,Z 280.148,A -85,B 0,C 180,E1 -24604.863,E2 -24604.863} C_VEL
LIN {X 0,Y 163.313,Z 271.974,A -85,B 0,C 180,E1 -24607.047,E2 -24607.047} C_VEL
LIN {X 0,Y 166.549,Z 263.467,A -85,B 0,C 180,E1 -24608.88,E2 -24608.88} C_VEL
LIN {X 0,Y 167.264,Z 261.528,A -85,B 0,C 180,E1 -24609.238,E2 -24609.238} C_VEL
LIN {X 0,Y 168.559,Z 256.591,A -85,B 0,C 180,E1 -24610.227,E2 -24610.227} C_VEL
LIN {X 0,Y 168.926,Z 248.253,A -85,B 0,C 180,E1 -24612.069,E2 -24612.069} C_VEL
LIN {X 0,Y 169.061,Z 239.627,A -85,B 0,C 180,E1 -24613.747,E2 -24613.747} C_VEL
LIN {X 0,Y 169.705,Z 234.127,A -85,B 0,C 180,E1 -24614.432,E2 -24614.432} C_VEL
LIN {X 0,Y 171.538,Z 224.179,A -85,B 0,C 180,E1 -24615.198,E2 -24615.198} C_VEL
LIN {X 0,Y 172.782,Z 214.448,A -85,B 0,C 180,E1 -24615.731,E2 -24615.731} C_VEL
LIN {X 0,Y 175.238,Z 179.663,A -85,B 0,C 180,E1 -24617.014,E2 -24617.014} C_VEL
LIN {X 0,Y 174.611,Z 176.65,A -85,B 0,C 180,E1 -24617.413,E2 -24617.413} C_VEL
LIN {X 0,Y 169.799,Z 163.903,A -85,B 0,C 180,E1 -24620.01,E2 -24620.01} C_VEL
LIN {X 0,Y 164.472,Z 152.458,A -85,B 0,C 180,E1 -24623.064,E2 -24623.064} C_VEL
LIN {X 0,Y 160.327,Z 144.605,A -85,B 0,C 180,E1 -24625.671,E2 -24625.671} C_VEL
LIN {X 0,Y 158.317,Z 141.265,A -85,B 0,C 180,E1 -24627.014,E2 -24627.014} C_VEL
LIN {X 0,Y 156.05,Z 138.032,A -85,B 0,C 180,E1 -24628.586,E2 -24628.586} C_VEL
LIN {X 0,Y 153.394,Z 134.262,A -85,B 0,C 180,E1 -24630.585,E2 -24630.585} C_VEL
LIN {X 0,Y 150.655,Z 130.706,A -85,B 0,C 180,E1 -24632.834,E2 -24632.834} C_VEL
LIN {X 0,Y 149.837,Z 129.592,A -85,B 0,C 180,E1 -24633.561,E2 -24633.561} C_VEL
LIN {X 0,Y 147.244,Z 126.83,A -85,B 0,C 180,E1 -24635.969,E2 -24635.969} C_VEL
LIN {X 0,Y 145.999,Z 124.65,A -85,B 0,C 180,E1 -24637.349,E2 -24637.349} C_VEL
LIN {X 0,Y 143.367,Z 122.472,A -85,B 0,C 180,E1 -24640.303,E2 -24640.303} C_VEL
LIN {X 0,Y 141.515,Z 119.207,A -85,B 0,C 180,E1 -24643.035,E2 -24643.035} C_VEL
LIN {X 0,Y 138.373,Z 116.892,A -85,B 0,C 180,E1 -24648.501,E2 -24648.501} C_VEL
LIN {X 0,Y 136.743,Z 113.747,A -85,B 0,C 180,E1 -24654.468,E2 -24654.468} C_VEL
LIN {X 0,Y 137.134,Z 112.969,A -85,B 0,C 180,E1 -24659.998,E2 -24659.998} C_VEL
LIN {X 0,Y 136.7,Z 113.585,A -85,B 0,C 180,E1 -24665.16,E2 -24665.16} C_VEL
LIN {X 0,Y 137.325,Z 115.307,A -85,B 0,C 180,E1 -24669.016,E2 -24669.016} C_VEL
LIN {X 0,Y 139.719,Z 118.194,A -85,B 0,C 180,E1 -24674.565,E2 -24674.565} C_VEL
LIN {X 0,Y 141.739,Z 119.478,A -85,B 0,C 180,E1 -24677.678,E2 -24677.678} C_VEL
LIN {X 0,Y 143.362,Z 122.468,A -85,B 0,C 180,E1 -24680.068,E2 -24680.068} C_VEL
LIN {X 0,Y 145.675,Z 124.466,A -85,B 0,C 180,E1 -24682.701,E2 -24682.701} C_VEL
LIN {X 0,Y 146.357,Z 125.236,A -85,B 0,C 180,E1 -24683.43,E2 -24683.43} C_VEL
LIN {X 0,Y 148.664,Z 128.606,A -85,B 0,C 180,E1 -24685.793,E2 -24685.793} C_VEL
LIN {X 0,Y 150.449,Z 130.335,A -85,B 0,C 180,E1 -24687.355,E2 -24687.355} C_VEL
LIN {X 0,Y 152.952,Z 133.818,A -85,B 0,C 180,E1 -24689.457,E2 -24689.457} C_VEL
LIN {X 0,Y 154.232,Z 135.432,A -85,B 0,C 180,E1 -24690.441,E2 -24690.441} C_VEL
LIN {X 0,Y 157.857,Z 140.554,A -85,B 0,C 180,E1 -24693.049,E2 -24693.049} C_VEL
LIN {X 0,Y 162.475,Z 147.378,A -85,B 0,C 180,E1 -24695.999,E2 -24695.999} C_VEL
LIN {X 0,Y 168.73,Z 157.596,A -85,B 0,C 180,E1 -24699.523,E2 -24699.523} C_VEL
LIN {X 0,Y 174.853,Z 169.32,A -85,B 0,C 180,E1 -24702.615,E2 -24702.615} C_VEL
LIN {X 0,Y 180.329,Z 181.939,A -85,B 0,C 180,E1 -24705.187,E2 -24705.187} C_VEL
LIN {X 0,Y 187.901,Z 199.881,A -85,B 0,C 180,E1 -24708.359,E2 -24708.359} C_VEL
LIN {X 0,Y 195.187,Z 213.865,A -85,B 0,C 180,E1 -24711.134,E2 -24711.134} C_VEL
LIN {X 0,Y 201.338,Z 224.63,A -85,B 0,C 180,E1 -24713.601,E2 -24713.601} C_VEL
LIN {X 0,Y 208.558,Z 235.359,A -85,B 0,C 180,E1 -24716.423,E2 -24716.423} C_VEL
LIN {X 0,Y 216.477,Z 245.37,A -85,B 0,C 180,E1 -24719.352,E2 -24719.352} C_VEL
LIN {X 0,Y 225.744,Z 255.317,A -85,B 0,C 180,E1 -24722.529,E2 -24722.529} C_VEL
LIN {X 0,Y 235.537,Z 263.765,A -85,B 0,C 180,E1 -24725.51,E2 -24725.51} C_VEL
LIN {X 0,Y 248.428,Z 272.903,A -85,B 0,C 180,E1 -24728.995,E2 -24728.995} C_VEL
LIN {X 0,Y 262.801,Z 281.413,A -85,B 0,C 180,E1 -24732.492,E2 -24732.492} C_VEL
LIN {X 0,Y 273.566,Z 287.556,A -85,B 0,C 180,E1 -24735.114,E2 -24735.114} C_VEL
LIN {X 0,Y 281.162,Z 292.076,A -85,B 0,C 180,E1 -24737.119,E2 -24737.119} C_VEL
LIN {X 0,Y 289.29,Z 296.984,A -85,B 0,C 180,E1 -24739.511,E2 -24739.511} C_VEL
LIN {X 0,Y 292.153,Z 298.759,A -85,B 0,C 180,E1 -24740.497,E2 -24740.497} C_VEL
LIN {X 0,Y 295.139,Z 300.86,A -85,B 0,C 180,E1 -24741.786,E2 -24741.786} C_VEL
LIN {X 0,Y 298.171,Z 302.816,A -85,B 0,C 180,E1 -24743.232,E2 -24743.232} C_VEL
LIN {X 0,Y 300.659,Z 304.174,A -85,B 0,C 180,E1 -24744.635,E2 -24744.635} C_VEL
LIN {X 0,Y 302.901,Z 305.25,A -85,B 0,C 180,E1 -24746.1,E2 -24746.1} C_VEL
LIN {X 0,Y 304.379,Z 305.899,A -85,B 0,C 180,E1 -24747.353,E2 -24747.353} C_VEL
LIN {X 0,Y 305.347,Z 306.289,A -85,B 0,C 180,E1 -24748.681,E2 -24748.681} C_VEL
LIN {X 0,Y 305.729,Z 306.397,A -85,B 0,C 180,E1 -24750,E2 -24750} C_VEL
LIN {X 0,Y 305.369,Z 306.288,A -85,B 0,C 180,E1 -24751.319,E2 -24751.319} C_VEL
LIN {X 0,Y 304.376,Z 305.907,A -85,B 0,C 180,E1 -24752.647,E2 -24752.647} C_VEL
LIN {X 0,Y 302.762,Z 305.213,A -85,B 0,C 180,E1 -24753.993,E2 -24753.993} C_VEL
LIN {X 0,Y 300.652,Z 304.204,A -85,B 0,C 180,E1 -24755.365,E2 -24755.365} C_VEL
LIN {X 0,Y 297.454,Z 302.405,A -85,B 0,C 180,E1 -24757.102,E2 -24757.102} C_VEL
LIN {X 0,Y 293.713,Z 299.867,A -85,B 0,C 180,E1 -24758.843,E2 -24758.843} C_VEL
LIN {X 0,Y 291.557,Z 298.393,A -85,B 0,C 180,E1 -24759.714,E2 -24759.714} C_VEL
LIN {X 0,Y 286.591,Z 295.347,A -85,B 0,C 180,E1 -24761.314,E2 -24761.314} C_VEL
LIN {X 0,Y 278.167,Z 290.241,A -85,B 0,C 180,E1 -24763.703,E2 -24763.703} C_VEL
LIN {X 0,Y 270.135,Z 285.655,A -85,B 0,C 180,E1 -24765.72,E2 -24765.72} C_VEL
LIN {X 0,Y 259.167,Z 279.407,A -85,B 0,C 180,E1 -24768.359,E2 -24768.359} C_VEL
LIN {X 0,Y 244.889,Z 270.619,A -85,B 0,C 180,E1 -24771.906,E2 -24771.906} C_VEL
LIN {X 0,Y 233.04,Z 261.759,A -85,B 0,C 180,E1 -24775.215,E2 -24775.215} C_VEL
LIN {X 0,Y 223.388,Z 252.953,A -85,B 0,C 180,E1 -24778.251,E2 -24778.251} C_VEL
LIN {X 0,Y 214.243,Z 242.663,A -85,B 0,C 180,E1 -24781.473,E2 -24781.473} C_VEL
LIN {X 0,Y 205.437,Z 230.826,A -85,B 0,C 180,E1 -24784.813,E2 -24784.813} C_VEL
LIN {X 0,Y 198.822,Z 220.354,A -85,B 0,C 180,E1 -24787.419,E2 -24787.419} C_VEL
LIN {X 0,Y 192.599,Z 209.03,A -85,B 0,C 180,E1 -24789.878,E2 -24789.878} C_VEL
LIN {X 0,Y 186.488,Z 196.764,A -85,B 0,C 180,E1 -24792.189,E2 -24792.189} C_VEL
LIN {X 0,Y 177.47,Z 175.118,A -85,B 0,C 180,E1 -24796.135,E2 -24796.135} C_VEL
LIN {X 0,Y 172.594,Z 164.728,A -85,B 0,C 180,E1 -24798.495,E2 -24798.495} C_VEL
LIN {X 0,Y 167.214,Z 155.065,A -85,B 0,C 180,E1 -24801.286,E2 -24801.286} C_VEL
LIN {X 0,Y 161.668,Z 146.125,A -85,B 0,C 180,E1 -24804.494,E2 -24804.494} C_VEL
LIN {X 0,Y 156.419,Z 138.442,A -85,B 0,C 180,E1 -24807.955,E2 -24807.955} C_VEL
LIN {X 0,Y 153.289,Z 134.191,A -85,B 0,C 180,E1 -24810.284,E2 -24810.284} C_VEL
LIN {X 0,Y 150.614,Z 130.654,A -85,B 0,C 180,E1 -24812.492,E2 -24812.492} C_VEL
LIN {X 0,Y 149.799,Z 129.581,A -85,B 0,C 180,E1 -24813.214,E2 -24813.214} C_VEL
LIN {X 0,Y 147.24,Z 126.814,A -85,B 0,C 180,E1 -24815.597,E2 -24815.597} C_VEL
LIN {X 0,Y 145.994,Z 124.64,A -85,B 0,C 180,E1 -24816.977,E2 -24816.977} C_VEL
LIN {X 0,Y 143.435,Z 122.57,A -85,B 0,C 180,E1 -24819.837,E2 -24819.837} C_VEL
LIN {X 0,Y 141.844,Z 119.713,A -85,B 0,C 180,E1 -24822.149,E2 -24822.149} C_VEL
LIN {X 0,Y 140.805,Z 118.777,A -85,B 0,C 180,E1 -24823.696,E2 -24823.696} C_VEL
LIN {X 0,Y 138.392,Z 116.978,A -85,B 0,C 180,E1 -24828.064,E2 -24828.064} C_VEL
LIN {X 0,Y 136.743,Z 113.871,A -85,B 0,C 180,E1 -24833.824,E2 -24833.824} C_VEL
LIN {X 0,Y 136.939,Z 113.072,A -85,B 0,C 180,E1 -24838.531,E2 -24838.531} C_VEL
LIN {X 0,Y 137.031,Z 113.005,A -85,B 0,C 180,E1 -24840.736,E2 -24840.736} C_VEL
LIN {X 0,Y 136.749,Z 113.837,A -85,B 0,C 180,E1 -24845.716,E2 -24845.716} C_VEL
LIN {X 0,Y 139.723,Z 118.205,A -85,B 0,C 180,E1 -24854.196,E2 -24854.196} C_VEL
LIN {X 0,Y 141.688,Z 119.402,A -85,B 0,C 180,E1 -24857.223,E2 -24857.223} C_VEL
LIN {X 0,Y 143.237,Z 122.308,A -85,B 0,C 180,E1 -24859.529,E2 -24859.529} C_VEL
LIN {X 0,Y 145.739,Z 124.513,A -85,B 0,C 180,E1 -24862.39,E2 -24862.39} C_VEL
LIN {X 0,Y 146.358,Z 125.278,A -85,B 0,C 180,E1 -24863.059,E2 -24863.059} C_VEL
LIN {X 0,Y 148.454,Z 128.375,A -85,B 0,C 180,E1 -24865.22,E2 -24865.22} C_VEL
LIN {X 0,Y 150.403,Z 130.259,A -85,B 0,C 180,E1 -24866.935,E2 -24866.935} C_VEL
LIN {X 0,Y 153.039,Z 133.943,A -85,B 0,C 180,E1 -24869.15,E2 -24869.15} C_VEL
LIN {X 0,Y 154.251,Z 135.472,A -85,B 0,C 180,E1 -24870.08,E2 -24870.08} C_VEL
LIN {X 0,Y 157.878,Z 140.598,A -85,B 0,C 180,E1 -24872.687,E2 -24872.687} C_VEL
LIN {X 0,Y 160.059,Z 144.13,A -85,B 0,C 180,E1 -24874.152,E2 -24874.152} C_VEL
LIN {X 0,Y 164.812,Z 153.079,A -85,B 0,C 180,E1 -24877.136,E2 -24877.136} C_VEL
LIN {X 0,Y 170.634,Z 165.862,A -85,B 0,C 180,E1 -24880.445,E2 -24880.445} C_VEL
LIN {X 0,Y 174.96,Z 177.745,A -85,B 0,C 180,E1 -24882.776,E2 -24882.776} C_VEL
LIN {X 0,Y 175.243,Z 179.609,A -85,B 0,C 180,E1 -24882.984,E2 -24882.984} C_VEL
LIN {X 0,Y 172.683,Z 215.618,A -85,B 0,C 180,E1 -24884.319,E2 -24884.319} C_VEL
LIN {X 0,Y 170.938,Z 228.226,A -85,B 0,C 180,E1 -24885.082,E2 -24885.082} C_VEL
LIN {X 0,Y 167.921,Z 241.794,A -85,B 0,C 180,E1 -24886.324,E2 -24886.324} C_VEL
LIN {X 0,Y 165.204,Z 251.304,A -85,B 0,C 180,E1 -24887.519,E2 -24887.519} C_VEL
LIN {X 0,Y 162.141,Z 260.577,A -85,B 0,C 180,E1 -24889.035,E2 -24889.035} C_VEL
LIN {X 0,Y 158.644,Z 269.515,A -85,B 0,C 180,E1 -24890.855,E2 -24890.855} C_VEL
LIN {X 0,Y 154.887,Z 278.038,A -85,B 0,C 180,E1 -24893.043,E2 -24893.043} C_VEL
LIN {X 0,Y 151.434,Z 285.253,A -85,B 0,C 180,E1 -24895.353,E2 -24895.353} C_VEL
LIN {X 0,Y 148.253,Z 291.452,A -85,B 0,C 180,E1 -24897.771,E2 -24897.771} C_VEL
LIN {X 0,Y 144.758,Z 297.989,A -85,B 0,C 180,E1 -24900.955,E2 -24900.955} C_VEL
LIN {X 0,Y 142.335,Z 302.493,A -85,B 0,C 180,E1 -24903.616,E2 -24903.616} C_VEL
LIN {X 0,Y 139.063,Z 307.984,A -85,B 0,C 180,E1 -24907.726,E2 -24907.726} C_VEL
LIN {X 0,Y 136.465,Z 312.308,A -85,B 0,C 180,E1 -24912.001,E2 -24912.001} C_VEL
LIN {X 0,Y 135.31,Z 314.682,A -85,B 0,C 180,E1 -24914.948,E2 -24914.948} C_VEL
LIN {X 0,Y 134.428,Z 316.487,A -85,B 0,C 180,E1 -24917.929,E2 -24917.929} C_VEL
LIN {X 0,Y 133.542,Z 318.947,A -85,B 0,C 180,E1 -24923.958,E2 -24923.958} C_VEL
LIN {X 0,Y 133.414,Z 319.541,A -85,B 0,C 180,E1 -24926.98,E2 -24926.98} C_VEL
LIN {X 0,Y 133.535,Z 319.702,A -85,B 0,C 180,E1 -24930,E2 -24930} C_VEL
LIN {X 0,Y 133.401,Z 319.541,A -85,B 0,C 180,E1 -24933.02,E2 -24933.02} C_VEL
LIN {X 0,Y 133.473,Z 318.945,A -85,B 0,C 180,E1 -24936.045,E2 -24936.045} C_VEL
LIN {X 0,Y 134.428,Z 316.487,A -85,B 0,C 180,E1 -24942.071,E2 -24942.071} C_VEL
LIN {X 0,Y 135.846,Z 313.528,A -85,B 0,C 180,E1 -24946.532,E2 -24946.532} C_VEL
LIN {X 0,Y 138.114,Z 309.537,A -85,B 0,C 180,E1 -24950.867,E2 -24950.867} C_VEL
LIN {X 0,Y 141.12,Z 304.407,A -85,B 0,C 180,E1 -24955.044,E2 -24955.044} C_VEL
LIN {X 0,Y 144.185,Z 299.157,A -85,B 0,C 180,E1 -24958.368,E2 -24958.368} C_VEL
LIN {X 0,Y 147.534,Z 292.828,A -85,B 0,C 180,E1 -24961.601,E2 -24961.601} C_VEL
LIN {X 0,Y 150.625,Z 286.879,A -85,B 0,C 180,E1 -24964.049,E2 -24964.049} C_VEL
LIN {X 0,Y 154.05,Z 279.957,A -85,B 0,C 180,E1 -24966.376,E2 -24966.376} C_VEL
LIN {X 0,Y 157.69,Z 271.783,A -85,B 0,C 180,E1 -24968.606,E2 -24968.606} C_VEL
LIN {X 0,Y 161.086,Z 263.276,A -85,B 0,C 180,E1 -24970.465,E2 -24970.465} C_VEL
LIN {X 0,Y 164.153,Z 254.566,A -85,B 0,C 180,E1 -24971.987,E2 -24971.987} C_VEL
LIN {X 0,Y 167.105,Z 244.814,A -85,B 0,C 180,E1 -24973.319,E2 -24973.319} C_VEL
LIN {X 0,Y 169.575,Z 234.737,A -85,B 0,C 180,E1 -24974.377,E2 -24974.377} C_VEL
LIN {X 0,Y 169.705,Z 234.127,A -85,B 0,C 180,E1 -24974.432,E2 -24974.432} C_VEL
LIN {X 0,Y 170.441,Z 228.545,A -85,B 0,C 180,E1 -24975.045,E2 -24975.045} C_VEL
LIN {X 0,Y 169.875,Z 219.4,A -85,B 0,C 180,E1 -24976.328,E2 -24976.328} C_VEL
LIN {X 0,Y 168.819,Z 210.116,A -85,B 0,C 180,E1 -24977.472,E2 -24977.472} C_VEL
LIN {X 0,Y 168.755,Z 204.311,A -85,B 0,C 180,E1 -24977.865,E2 -24977.865} C_VEL
LIN {X 0,Y 170.387,Z 180.949,A -85,B 0,C 180,E1 -24978.702,E2 -24978.702} C_VEL
LIN {X 0,Y 166.231,Z 169.27,A -85,B 0,C 180,E1 -24981.127,E2 -24981.127} C_VEL
LIN {X 0,Y 161.404,Z 158.315,A -85,B 0,C 180,E1 -24984.092,E2 -24984.092} C_VEL
LIN {X 0,Y 157.417,Z 150.37,A -85,B 0,C 180,E1 -24986.772,E2 -24986.772} C_VEL
LIN {X 0,Y 155.133,Z 146.435,A -85,B 0,C 180,E1 -24988.41,E2 -24988.41} C_VEL
LIN {X 0,Y 151.099,Z 140.534,A -85,B 0,C 180,E1 -24991.54,E2 -24991.54} C_VEL
LIN {X 0,Y 147.619,Z 135.896,A -85,B 0,C 180,E1 -24994.627,E2 -24994.627} C_VEL
LIN {X 0,Y 144.838,Z 132.453,A -85,B 0,C 180,E1 -24997.463,E2 -24997.463} C_VEL
LIN {X 0,Y 144.28,Z 131.308,A -85,B 0,C 180,E1 -24998.146,E2 -24998.146} C_VEL
LIN {X 0,Y 141.732,Z 129.014,A -85,B 0,C 180,E1 -25001.196,E2 -25001.196} C_VEL
LIN {X 0,Y 139.972,Z 125.886,A -85,B 0,C 180,E1 -25003.968,E2 -25003.968} C_VEL
LIN {X 0,Y 137.409,Z 124.01,A -85,B 0,C 180,E1 -25008.645,E2 -25008.645} C_VEL
LIN {X 0,Y 135.567,Z 120.617,A -85,B 0,C 180,E1 -25015.166,E2 -25015.166} C_VEL
LIN {X 0,Y 135.148,Z 119.794,A -85,B 0,C 180,E1 -25019.998,E2 -25019.998} C_VEL
LIN {X 0,Y 135.627,Z 120.769,A -85,B 0,C 180,E1 -25025.574,E2 -25025.574} C_VEL
LIN {X 0,Y 138.572,Z 125.124,A -85,B 0,C 180,E1 -25034.126,E2 -25034.126} C_VEL
LIN {X 0,Y 140.237,Z 126.234,A -85,B 0,C 180,E1 -25036.84,E2 -25036.84} C_VEL
LIN {X 0,Y 141.976,Z 129.358,A -85,B 0,C 180,E1 -25039.518,E2 -25039.518} C_VEL
LIN {X 0,Y 144.46,Z 131.663,A -85,B 0,C 180,E1 -25042.453,E2 -25042.453} C_VEL
LIN {X 0,Y 146.771,Z 135.1,A -85,B 0,C 180,E1 -25044.958,E2 -25044.958} C_VEL
LIN {X 0,Y 148.395,Z 136.845,A -85,B 0,C 180,E1 -25046.471,E2 -25046.471} C_VEL
LIN {X 0,Y 151.114,Z 140.539,A -85,B 0,C 180,E1 -25048.848,E2 -25048.848} C_VEL
LIN {X 0,Y 155.186,Z 146.512,A -85,B 0,C 180,E1 -25052.006,E2 -25052.006} C_VEL
LIN {X 0,Y 159.194,Z 152.546,A -85,B 0,C 180,E1 -25054.733,E2 -25054.733} C_VEL
LIN {X 0,Y 165.405,Z 163.138,A -85,B 0,C 180,E1 -25058.478,E2 -25058.478} C_VEL
LIN {X 0,Y 170.781,Z 173.772,A -85,B 0,C 180,E1 -25061.378,E2 -25061.378} C_VEL
LIN {X 0,Y 176.142,Z 186.575,A -85,B 0,C 180,E1 -25064.075,E2 -25064.075} C_VEL
LIN {X 0,Y 183.381,Z 204.236,A -85,B 0,C 180,E1 -25067.335,E2 -25067.335} C_VEL
LIN {X 0,Y 189.107,Z 216.06,A -85,B 0,C 180,E1 -25069.833,E2 -25069.833} C_VEL
LIN {X 0,Y 194.374,Z 225.914,A -85,B 0,C 180,E1 -25072.209,E2 -25072.209} C_VEL
LIN {X 0,Y 200.108,Z 235.223,A -85,B 0,C 180,E1 -25074.74,E2 -25074.74} C_VEL
LIN {X 0,Y 206.435,Z 244.15,A -85,B 0,C 180,E1 -25077.413,E2 -25077.413} C_VEL
LIN {X 0,Y 213.145,Z 252.329,A -85,B 0,C 180,E1 -25080.07,E2 -25080.07} C_VEL
LIN {X 0,Y 220.984,Z 260.474,A -85,B 0,C 180,E1 -25082.932,E2 -25082.932} C_VEL
LIN {X 0,Y 232.088,Z 269.538,A -85,B 0,C 180,E1 -25086.458,E2 -25086.458} C_VEL
LIN {X 0,Y 240.929,Z 275.625,A -85,B 0,C 180,E1 -25088.977,E2 -25088.977} C_VEL
LIN {X 0,Y 253.813,Z 283.048,A -85,B 0,C 180,E1 -25092.267,E2 -25092.267} C_VEL
LIN {X 0,Y 262.831,Z 287.851,A -85,B 0,C 180,E1 -25094.491,E2 -25094.491} C_VEL
LIN {X 0,Y 270.697,Z 292.026,A -85,B 0,C 180,E1 -25096.487,E2 -25096.487} C_VEL
LIN {X 0,Y 279.285,Z 296.794,A -85,B 0,C 180,E1 -25098.929,E2 -25098.929} C_VEL
LIN {X 0,Y 284.872,Z 299.872,A -85,B 0,C 180,E1 -25100.685,E2 -25100.685} C_VEL
LIN {X 0,Y 288.727,Z 302.397,A -85,B 0,C 180,E1 -25102.306,E2 -25102.306} C_VEL
LIN {X 0,Y 293.049,Z 305.028,A -85,B 0,C 180,E1 -25104.495,E2 -25104.495} C_VEL
LIN {X 0,Y 295.82,Z 306.44,A -85,B 0,C 180,E1 -25106.206,E2 -25106.206} C_VEL
LIN {X 0,Y 297.139,Z 307.048,A -85,B 0,C 180,E1 -25107.289,E2 -25107.289} C_VEL
LIN {X 0,Y 298.27,Z 307.463,A -85,B 0,C 180,E1 -25108.65,E2 -25108.65} C_VEL
LIN {X 0,Y 298.732,Z 307.581,A -85,B 0,C 180,E1 -25110,E2 -25110} C_VEL
LIN {X 0,Y 298.286,Z 307.467,A -85,B 0,C 180,E1 -25111.35,E2 -25111.35} C_VEL
LIN {X 0,Y 297.133,Z 307.062,A -85,B 0,C 180,E1 -25112.711,E2 -25112.711} C_VEL
LIN {X 0,Y 295.335,Z 306.258,A -85,B 0,C 180,E1 -25114.094,E2 -25114.094} C_VEL
LIN {X 0,Y 293.04,Z 305.035,A -85,B 0,C 180,E1 -25115.505,E2 -25115.505} C_VEL
LIN {X 0,Y 290.278,Z 303.434,A -85,B 0,C 180,E1 -25116.953,E2 -25116.953} C_VEL
LIN {X 0,Y 287.011,Z 301.282,A -85,B 0,C 180,E1 -25118.449,E2 -25118.449} C_VEL
LIN {X 0,Y 282.707,Z 298.66,A -85,B 0,C 180,E1 -25120.021,E2 -25120.021} C_VEL
LIN {X 0,Y 277.114,Z 295.608,A -85,B 0,C 180,E1 -25121.706,E2 -25121.706} C_VEL
LIN {X 0,Y 270.654,Z 292.027,A -85,B 0,C 180,E1 -25123.515,E2 -25123.515} C_VEL
LIN {X 0,Y 261.027,Z 286.94,A -85,B 0,C 180,E1 -25125.952,E2 -25125.952} C_VEL
LIN {X 0,Y 246.256,Z 278.767,A -85,B 0,C 180,E1 -25129.647,E2 -25129.647} C_VEL
LIN {X 0,Y 233.977,Z 270.927,A -85,B 0,C 180,E1 -25132.984,E2 -25132.984} C_VEL
LIN {X 0,Y 224.028,Z 263.149,A -85,B 0,C 180,E1 -25136.052,E2 -25136.052} C_VEL
LIN {X 0,Y 215.121,Z 254.495,A -85,B 0,C 180,E1 -25139.18,E2 -25139.18} C_VEL
LIN {X 0,Y 207.514,Z 245.514,A -85,B 0,C 180,E1 -25142.149,E2 -25142.149} C_VEL
LIN {X 0,Y 201.151,Z 236.757,A -85,B 0,C 180,E1 -25144.811,E2 -25144.811} C_VEL
LIN {X 0,Y 195.972,Z 228.722,A -85,B 0,C 180,E1 -25147.069,E2 -25147.069} C_VEL
LIN {X 0,Y 190.129,Z 218.027,A -85,B 0,C 180,E1 -25149.709,E2 -25149.709} C_VEL
LIN {X 0,Y 184.596,Z 206.756,A -85,B 0,C 180,E1 -25152.166,E2 -25152.166} C_VEL
LIN {X 0,Y 177.726,Z 190.866,A -85,B 0,C 180,E1 -25155.154,E2 -25155.154} C_VEL
LIN {X 0,Y 172.935,Z 178.699,A -85,B 0,C 180,E1 -25157.515,E2 -25157.515} C_VEL
LIN {X 0,Y 168.615,Z 169.336,A -85,B 0,C 180,E1 -25159.757,E2 -25159.757} C_VEL
LIN {X 0,Y 163.9,Z 160.507,A -85,B 0,C 180,E1 -25162.379,E2 -25162.379} C_VEL
LIN {X 0,Y 158.761,Z 151.912,A -85,B 0,C 180,E1 -25165.544,E2 -25165.544} C_VEL
LIN {X 0,Y 153.861,Z 144.465,A -85,B 0,C 180,E1 -25168.981,E2 -25168.981} C_VEL
LIN {X 0,Y 150.738,Z 140.135,A -85,B 0,C 180,E1 -25171.454,E2 -25171.454} C_VEL
LIN {X 0,Y 147.837,Z 136.091,A -85,B 0,C 180,E1 -25174.052,E2 -25174.052} C_VEL
LIN {X 0,Y 145.216,Z 133.057,A -85,B 0,C 180,E1 -25176.658,E2 -25176.658} C_VEL
LIN {X 0,Y 144.183,Z 131.281,A -85,B 0,C 180,E1 -25177.868,E2 -25177.868} C_VEL
LIN {X 0,Y 141.697,Z 128.973,A -85,B 0,C 180,E1 -25180.865,E2 -25180.865} C_VEL
LIN {X 0,Y 139.967,Z 125.891,A -85,B 0,C 180,E1 -25183.596,E2 -25183.596} C_VEL
LIN {X 0,Y 137.341,Z 123.973,A -85,B 0,C 180,E1 -25188.417,E2 -25188.417} C_VEL
LIN {X 0,Y 135.627,Z 120.767,A -85,B 0,C 180,E1 -25194.426,E2 -25194.426} C_VEL
LIN {X 0,Y 135.151,Z 119.774,A -85,B 0,C 180,E1 -25200.002,E2 -25200.002} C_VEL
LIN {X 0,Y 135.631,Z 120.745,A -85,B 0,C 180,E1 -25205.204,E2 -25205.204} C_VEL
LIN {X 0,Y 138.675,Z 125.188,A -85,B 0,C 180,E1 -25213.931,E2 -25213.931} C_VEL
LIN {X 0,Y 140.193,Z 126.117,A -85,B 0,C 180,E1 -25216.38,E2 -25216.38} C_VEL
LIN {X 0,Y 141.86,Z 129.147,A -85,B 0,C 180,E1 -25218.974,E2 -25218.974} C_VEL
LIN {X 0,Y 144.445,Z 131.712,A -85,B 0,C 180,E1 -25222.067,E2 -25222.067} C_VEL
LIN {X 0,Y 146.94,Z 135.268,A -85,B 0,C 180,E1 -25224.742,E2 -25224.742} C_VEL
LIN {X 0,Y 148.389,Z 136.854,A -85,B 0,C 180,E1 -25226.09,E2 -25226.09} C_VEL
LIN {X 0,Y 152.074,Z 142.009,A -85,B 0,C 180,E1 -25229.264,E2 -25229.264} C_VEL
LIN {X 0,Y 155.033,Z 146.284,A -85,B 0,C 180,E1 -25231.518,E2 -25231.518} C_VEL
LIN {X 0,Y 157.65,Z 150.76,A -85,B 0,C 180,E1 -25233.388,E2 -25233.388} C_VEL
LIN {X 0,Y 161.835,Z 159.21,A -85,B 0,C 180,E1 -25236.182,E2 -25236.182} C_VEL
LIN {X 0,Y 166.684,Z 170.338,A -85,B 0,C 180,E1 -25239.136,E2 -25239.136} C_VEL
LIN {X 0,Y 170.393,Z 180.888,A -85,B 0,C 180,E1 -25241.296,E2 -25241.296} C_VEL
LIN {X 0,Y 167.809,Z 215.317,A -85,B 0,C 180,E1 -25242.577,E2 -25242.577} C_VEL
LIN {X 0,Y 166.038,Z 227.75,A -85,B 0,C 180,E1 -25243.334,E2 -25243.334} C_VEL
LIN {X 0,Y 162.87,Z 241.604,A -85,B 0,C 180,E1 -25244.603,E2 -25244.603} C_VEL
LIN {X 0,Y 160.046,Z 251.114,A -85,B 0,C 180,E1 -25245.805,E2 -25245.805} C_VEL
LIN {X 0,Y 156.849,Z 260.386,A -85,B 0,C 180,E1 -25247.335,E2 -25247.335} C_VEL
LIN {X 0,Y 153.194,Z 269.325,A -85,B 0,C 180,E1 -25249.176,E2 -25249.176} C_VEL
LIN {X 0,Y 149.265,Z 277.847,A -85,B 0,C 180,E1 -25251.401,E2 -25251.401} C_VEL
LIN {X 0,Y 145.642,Z 285.062,A -85,B 0,C 180,E1 -25253.763,E2 -25253.763} C_VEL
LIN {X 0,Y 142.27,Z 291.26,A -85,B 0,C 180,E1 -25256.239,E2 -25256.239} C_VEL
LIN {X 0,Y 138.322,Z 298.181,A -85,B 0,C 180,E1 -25259.744,E2 -25259.744} C_VEL
LIN {X 0,Y 136.004,Z 302.303,A -85,B 0,C 180,E1 -25262.285,E2 -25262.285} C_VEL
LIN {X 0,Y 132.494,Z 307.792,A -85,B 0,C 180,E1 -25266.558,E2 -25266.558} C_VEL
LIN {X 0,Y 129.698,Z 312.117,A -85,B 0,C 180,E1 -25271.027,E2 -25271.027} C_VEL
LIN {X 0,Y 128.428,Z 314.49,A -85,B 0,C 180,E1 -25274.12,E2 -25274.12} C_VEL
LIN {X 0,Y 127.458,Z 316.295,A -85,B 0,C 180,E1 -25277.258,E2 -25277.258} C_VEL
LIN {X 0,Y 126.463,Z 318.756,A -85,B 0,C 180,E1 -25283.619,E2 -25283.619} C_VEL
LIN {X 0,Y 126.317,Z 319.351,A -85,B 0,C 180,E1 -25286.811,E2 -25286.811} C_VEL
LIN {X 0,Y 126.431,Z 319.511,A -85,B 0,C 180,E1 -25290,E2 -25290} C_VEL
LIN {X 0,Y 126.306,Z 319.35,A -85,B 0,C 180,E1 -25293.19,E2 -25293.19} C_VEL
LIN {X 0,Y 126.414,Z 318.754,A -85,B 0,C 180,E1 -25296.384,E2 -25296.384} C_VEL
LIN {X 0,Y 127.458,Z 316.295,A -85,B 0,C 180,E1 -25302.742,E2 -25302.742} C_VEL
LIN {X 0,Y 129.002,Z 313.336,A -85,B 0,C 180,E1 -25307.436,E2 -25307.436} C_VEL
LIN {X 0,Y 131.48,Z 309.346,A -85,B 0,C 180,E1 -25311.973,E2 -25311.973} C_VEL
LIN {X 0,Y 134.708,Z 304.216,A -85,B 0,C 180,E1 -25316.325,E2 -25316.325} C_VEL
LIN {X 0,Y 137.939,Z 298.956,A -85,B 0,C 180,E1 -25319.786,E2 -25319.786} C_VEL
LIN {X 0,Y 141.525,Z 292.637,A -85,B 0,C 180,E1 -25323.11,E2 -25323.11} C_VEL
LIN {X 0,Y 144.787,Z 286.688,A -85,B 0,C 180,E1 -25325.625,E2 -25325.625} C_VEL
LIN {X 0,Y 148.381,Z 279.766,A -85,B 0,C 180,E1 -25328.006,E2 -25328.006} C_VEL
LIN {X 0,Y 152.197,Z 271.592,A -85,B 0,C 180,E1 -25330.276,E2 -25330.276} C_VEL
LIN {X 0,Y 155.76,Z 263.086,A -85,B 0,C 180,E1 -25332.157,E2 -25332.157} C_VEL
LIN {X 0,Y 158.958,Z 254.376,A -85,B 0,C 180,E1 -25333.695,E2 -25333.695} C_VEL
LIN {X 0,Y 162.017,Z 244.623,A -85,B 0,C 180,E1 -25335.04,E2 -25335.04} C_VEL
LIN {X 0,Y 164.586,Z 234.546,A -85,B 0,C 180,E1 -25336.102,E2 -25336.102} C_VEL
LIN {X 0,Y 166.479,Z 224.796,A -85,B 0,C 180,E1 -25336.877,E2 -25336.877} C_VEL
LIN {X 0,Y 167.814,Z 215.215,A -85,B 0,C 180,E1 -25337.42,E2 -25337.42} C_VEL
LIN {X 0,Y 168.755,Z 204.311,A -85,B 0,C 180,E1 -25337.865,E2 -25337.865} C_VEL
LIN {X 0,Y 168.716,Z 198.486,A -85,B 0,C 180,E1 -25338.242,E2 -25338.242} C_VEL
LIN {X 0,Y 167.991,Z 192.875,A -85,B 0,C 180,E1 -25338.873,E2 -25338.873} C_VEL
LIN {X 0,Y 166.303,Z 185.76,A -85,B 0,C 180,E1 -25340.003,E2 -25340.003} C_VEL
LIN {X 0,Y 163.075,Z 175.652,A -85,B 0,C 180,E1 -25342.066,E2 -25342.066} C_VEL
LIN {X 0,Y 159.323,Z 166.281,A -85,B 0,C 180,E1 -25344.524,E2 -25344.524} C_VEL
LIN {X 0,Y 154.888,Z 156.641,A -85,B 0,C 180,E1 -25347.684,E2 -25347.684} C_VEL
LIN {X 0,Y 152.262,Z 151.962,A -85,B 0,C 180,E1 -25349.692,E2 -25349.692} C_VEL
LIN {X 0,Y 148.43,Z 146.288,A -85,B 0,C 180,E1 -25352.886,E2 -25352.886} C_VEL
LIN {X 0,Y 145.602,Z 142.304,A -85,B 0,C 180,E1 -25355.586,E2 -25355.586} C_VEL
LIN {X 0,Y 142.806,Z 138.553,A -85,B 0,C 180,E1 -25358.661,E2 -25358.661} C_VEL
LIN {X 0,Y 142.082,Z 137.62,A -85,B 0,C 180,E1 -25359.545,E2 -25359.545} C_VEL
LIN {X 0,Y 139.435,Z 134.439,A -85,B 0,C 180,E1 -25363.199,E2 -25363.199} C_VEL
LIN {X 0,Y 138.568,Z 132.692,A -85,B 0,C 180,E1 -25364.744,E2 -25364.744} C_VEL
LIN {X 0,Y 136.172,Z 130.695,A -85,B 0,C 180,E1 -25369.5,E2 -25369.5} C_VEL
LIN {X 0,Y 134.581,Z 127.504,A -85,B 0,C 180,E1 -25375.881,E2 -25375.881} C_VEL
LIN {X 0,Y 134.282,Z 126.848,A -85,B 0,C 180,E1 -25379.998,E2 -25379.998} C_VEL
LIN {X 0,Y 134.724,Z 127.824,A -85,B 0,C 180,E1 -25385.424,E2 -25385.424} C_VEL
LIN {X 0,Y 137.478,Z 132.084,A -85,B 0,C 180,E1 -25393.762,E2 -25393.762} C_VEL
LIN {X 0,Y 138.766,Z 132.999,A -85,B 0,C 180,E1 -25395.984,E2 -25395.984} C_VEL
LIN {X 0,Y 140.864,Z 136.518,A -85,B 0,C 180,E1 -25399.308,E2 -25399.308} C_VEL
LIN {X 0,Y 142.717,Z 138.321,A -85,B 0,C 180,E1 -25401.594,E2 -25401.594} C_VEL
LIN {X 0,Y 145.275,Z 141.968,A -85,B 0,C 180,E1 -25404.469,E2 -25404.469} C_VEL
LIN {X 0,Y 146.407,Z 143.411,A -85,B 0,C 180,E1 -25405.595,E2 -25405.595} C_VEL
LIN {X 0,Y 149.671,Z 148.096,A -85,B 0,C 180,E1 -25408.577,E2 -25408.577} C_VEL
LIN {X 0,Y 152.83,Z 152.831,A -85,B 0,C 180,E1 -25411.123,E2 -25411.123} C_VEL
LIN {X 0,Y 157.342,Z 160.129,A -85,B 0,C 180,E1 -25414.35,E2 -25414.35} C_VEL
LIN {X 0,Y 162.577,Z 169.495,A -85,B 0,C 180,E1 -25417.652,E2 -25417.652} C_VEL
LIN {X 0,Y 167.361,Z 179.502,A -85,B 0,C 180,E1 -25420.396,E2 -25420.396} C_VEL
LIN {X 0,Y 172.077,Z 191.455,A -85,B 0,C 180,E1 -25422.944,E2 -25422.944} C_VEL
LIN {X 0,Y 178.641,Z 208.104,A -85,B 0,C 180,E1 -25426.19,E2 -25426.19} C_VEL
LIN {X 0,Y 183.039,Z 217.814,A -85,B 0,C 180,E1 -25428.375,E2 -25428.375} C_VEL
LIN {X 0,Y 187.725,Z 227.385,A -85,B 0,C 180,E1 -25430.788,E2 -25430.788} C_VEL
LIN {X 0,Y 192.737,Z 236.459,A -85,B 0,C 180,E1 -25433.34,E2 -25433.34} C_VEL
LIN {X 0,Y 198.709,Z 245.645,A -85,B 0,C 180,E1 -25436.215,E2 -25436.215} C_VEL
LIN {X 0,Y 206.055,Z 254.981,A -85,B 0,C 180,E1 -25439.449,E2 -25439.449} C_VEL
LIN {X 0,Y 214.015,Z 263.44,A -85,B 0,C 180,E1 -25442.63,E2 -25442.63} C_VEL
LIN {X 0,Y 223.322,Z 271.3,A -85,B 0,C 180,E1 -25445.87,E2 -25445.87} C_VEL
LIN {X 0,Y 236.041,Z 279.837,A -85,B 0,C 180,E1 -25449.698,E2 -25449.698} C_VEL
LIN {X 0,Y 249.549,Z 287.108,A -85,B 0,C 180,E1 -25453.24,E2 -25453.24} C_VEL
LIN {X 0,Y 260.678,Z 292.577,A -85,B 0,C 180,E1 -25456.063,E2 -25456.063} C_VEL
LIN {X 0,Y 269.162,Z 296.77,A -85,B 0,C 180,E1 -25458.37,E2 -25458.37} C_VEL
LIN {X 0,Y 275.837,Z 300.124,A -85,B 0,C 180,E1 -25460.379,E2 -25460.379} C_VEL
LIN {X 0,Y 278.644,Z 301.51,A -85,B 0,C 180,E1 -25461.296,E2 -25461.296} C_VEL
LIN {X 0,Y 283.087,Z 304.121,A -85,B 0,C 180,E1 -25463.234,E2 -25463.234} C_VEL
LIN {X 0,Y 285.226,Z 305.375,A -85,B 0,C 180,E1 -25464.344,E2 -25464.344} C_VEL
LIN {X 0,Y 288.72,Z 307.141,A -85,B 0,C 180,E1 -25466.379,E2 -25466.379} C_VEL
LIN {X 0,Y 289.806,Z 307.606,A -85,B 0,C 180,E1 -25467.22,E2 -25467.22} C_VEL
LIN {X 0,Y 291.076,Z 308.112,A -85,B 0,C 180,E1 -25468.616,E2 -25468.616} C_VEL
LIN {X 0,Y 291.669,Z 308.263,A -85,B 0,C 180,E1 -25470,E2 -25470} C_VEL
LIN {X 0,Y 291.087,Z 308.115,A -85,B 0,C 180,E1 -25471.383,E2 -25471.383} C_VEL
LIN {X 0,Y 289.801,Z 307.607,A -85,B 0,C 180,E1 -25472.78,E2 -25472.78} C_VEL
LIN {X 0,Y 287.762,Z 306.691,A -85,B 0,C 180,E1 -25474.202,E2 -25474.202} C_VEL
LIN {X 0,Y 285.222,Z 305.375,A -85,B 0,C 180,E1 -25475.656,E2 -25475.656} C_VEL
LIN {X 0,Y 282.272,Z 303.661,A -85,B 0,C 180,E1 -25477.151,E2 -25477.151} C_VEL
LIN {X 0,Y 278.591,Z 301.511,A -85,B 0,C 180,E1 -25478.706,E2 -25478.706} C_VEL
LIN {X 0,Y 271.893,Z 298.168,A -85,B 0,C 180,E1 -25480.82,E2 -25480.82} C_VEL
LIN {X 0,Y 266.284,Z 295.344,A -85,B 0,C 180,E1 -25482.441,E2 -25482.441} C_VEL
LIN {X 0,Y 258.685,Z 291.635,A -85,B 0,C 180,E1 -25484.431,E2 -25484.431} C_VEL
LIN {X 0,Y 246.792,Z 285.72,A -85,B 0,C 180,E1 -25487.45,E2 -25487.45} C_VEL
LIN {X 0,Y 232.693,Z 277.781,A -85,B 0,C 180,E1 -25491.25,E2 -25491.25} C_VEL
LIN {X 0,Y 221.55,Z 269.937,A -85,B 0,C 180,E1 -25494.709,E2 -25494.709} C_VEL
LIN {X 0,Y 211.855,Z 261.326,A -85,B 0,C 180,E1 -25498.196,E2 -25498.196} C_VEL
LIN {X 0,Y 203.589,Z 251.97,A -85,B 0,C 180,E1 -25501.63,E2 -25501.63} C_VEL
LIN {X 0,Y 195.85,Z 241.289,A -85,B 0,C 180,E1 -25505.189,E2 -25505.189} C_VEL
LIN {X 0,Y 189.697,Z 231.117,A -85,B 0,C 180,E1 -25508.221,E2 -25508.221} C_VEL
LIN {X 0,Y 183.764,Z 219.358,A -85,B 0,C 180,E1 -25511.26,E2 -25511.26} C_VEL
LIN {X 0,Y 178.566,Z 207.792,A -85,B 0,C 180,E1 -25513.886,E2 -25513.886} C_VEL
LIN {X 0,Y 172.487,Z 192.546,A -85,B 0,C 180,E1 -25516.843,E2 -25516.843} C_VEL
LIN {X 0,Y 168.016,Z 181.076,A -85,B 0,C 180,E1 -25519.239,E2 -25519.239} C_VEL
LIN {X 0,Y 163.524,Z 171.385,A -85,B 0,C 180,E1 -25521.785,E2 -25521.785} C_VEL
LIN {X 0,Y 158.273,Z 161.685,A -85,B 0,C 180,E1 -25525.036,E2 -25525.036} C_VEL
LIN {X 0,Y 153.353,Z 153.637,A -85,B 0,C 180,E1 -25528.481,E2 -25528.481} C_VEL
LIN {X 0,Y 150.12,Z 148.807,A -85,B 0,C 180,E1 -25531.038,E2 -25531.038} C_VEL
LIN {X 0,Y 148.348,Z 146.202,A -85,B 0,C 180,E1 -25532.579,E2 -25532.579} C_VEL
LIN {X 0,Y 145.603,Z 142.285,A -85,B 0,C 180,E1 -25535.209,E2 -25535.209} C_VEL
LIN {X 0,Y 142.968,Z 138.828,A -85,B 0,C 180,E1 -25538.083,E2 -25538.083} C_VEL
LIN {X 0,Y 142.216,Z 137.746,A -85,B 0,C 180,E1 -25539.007,E2 -25539.007} C_VEL
LIN {X 0,Y 139.674,Z 134.873,A -85,B 0,C 180,E1 -25542.43,E2 -25542.43} C_VEL
LIN {X 0,Y 138.675,Z 132.763,A -85,B 0,C 180,E1 -25544.194,E2 -25544.194} C_VEL
LIN {X 0,Y 136.141,Z 130.729,A -85,B 0,C 180,E1 -25549.181,E2 -25549.181} C_VEL
LIN {X 0,Y 134.632,Z 127.646,A -85,B 0,C 180,E1 -25555.136,E2 -25555.136} C_VEL
LIN {X 0,Y 134.286,Z 126.816,A -85,B 0,C 180,E1 -25560.002,E2 -25560.002} C_VEL
LIN {X 0,Y 134.695,Z 127.746,A -85,B 0,C 180,E1 -25564.865,E2 -25564.865} C_VEL
LIN {X 0,Y 137.63,Z 132.171,A -85,B 0,C 180,E1 -25573.662,E2 -25573.662} C_VEL
LIN {X 0,Y 138.799,Z 132.992,A -85,B 0,C 180,E1 -25575.653,E2 -25575.653} C_VEL
LIN {X 0,Y 140.554,Z 136.089,A -85,B 0,C 180,E1 -25578.495,E2 -25578.495} C_VEL
LIN {X 0,Y 142.711,Z 138.366,A -85,B 0,C 180,E1 -25581.217,E2 -25581.217} C_VEL
LIN {X 0,Y 145.437,Z 142.149,A -85,B 0,C 180,E1 -25584.253,E2 -25584.253} C_VEL
LIN {X 0,Y 146.568,Z 143.66,A -85,B 0,C 180,E1 -25585.378,E2 -25585.378} C_VEL
LIN {X 0,Y 149.759,Z 148.236,A -85,B 0,C 180,E1 -25588.275,E2 -25588.275} C_VEL
LIN {X 0,Y 152.563,Z 152.455,A -85,B 0,C 180,E1 -25590.544,E2 -25590.544} C_VEL
LIN {X 0,Y 155.471,Z 157.887,A -85,B 0,C 180,E1 -25592.756,E2 -25592.756} C_VEL
LIN {X 0,Y 159.637,Z 166.993,A -85,B 0,C 180,E1 -25595.687,E2 -25595.687} C_VEL
LIN {X 0,Y 163.105,Z 175.69,A -85,B 0,C 180,E1 -25597.95,E2 -25597.95} C_VEL
LIN {X 0,Y 165.619,Z 183.024,A -85,B 0,C 180,E1 -25599.535,E2 -25599.535} C_VEL
LIN {X 0,Y 163.076,Z 215.309,A -85,B 0,C 180,E1 -25600.751,E2 -25600.751} C_VEL
LIN {X 0,Y 161.169,Z 228.085,A -85,B 0,C 180,E1 -25601.538,E2 -25601.538} C_VEL
LIN {X 0,Y 157.977,Z 241.414,A -85,B 0,C 180,E1 -25602.774,E2 -25602.774} C_VEL
LIN {X 0,Y 155.034,Z 250.923,A -85,B 0,C 180,E1 -25603.975,E2 -25603.975} C_VEL
LIN {X 0,Y 151.696,Z 260.196,A -85,B 0,C 180,E1 -25605.514,E2 -25605.514} C_VEL
LIN {X 0,Y 147.891,Z 269.134,A -85,B 0,C 180,E1 -25607.376,E2 -25607.376} C_VEL
LIN {X 0,Y 143.762,Z 277.656,A -85,B 0,C 180,E1 -25609.628,E2 -25609.628} C_VEL
LIN {X 0,Y 139.975,Z 284.871,A -85,B 0,C 180,E1 -25612.044,E2 -25612.044} C_VEL
LIN {X 0,Y 136.393,Z 291.069,A -85,B 0,C 180,E1 -25614.572,E2 -25614.572} C_VEL
LIN {X 0,Y 132.478,Z 297.607,A -85,B 0,C 180,E1 -25617.961,E2 -25617.961} C_VEL
LIN {X 0,Y 129.73,Z 302.111,A -85,B 0,C 180,E1 -25620.819,E2 -25620.819} C_VEL
LIN {X 0,Y 125.987,Z 307.601,A -85,B 0,C 180,E1 -25625.268,E2 -25625.268} C_VEL
LIN {X 0,Y 122.981,Z 311.926,A -85,B 0,C 180,E1 -25629.947,E2 -25629.947} C_VEL
LIN {X 0,Y 121.56,Z 314.298,A -85,B 0,C 180,E1 -25633.197,E2 -25633.197} C_VEL
LIN {X 0,Y 120.517,Z 316.104,A -85,B 0,C 180,E1 -25636.511,E2 -25636.511} C_VEL
LIN {X 0,Y 119.391,Z 318.565,A -85,B 0,C 180,E1 -25643.239,E2 -25643.239} C_VEL
LIN {X 0,Y 119.231,Z 319.16,A -85,B 0,C 180,E1 -25646.621,E2 -25646.621} C_VEL
LIN {X 0,Y 119.337,Z 319.321,A -85,B 0,C 180,E1 -25650,E2 -25650} C_VEL
LIN {X 0,Y 119.222,Z 319.16,A -85,B 0,C 180,E1 -25653.379,E2 -25653.379} C_VEL
LIN {X 0,Y 119.336,Z 318.563,A -85,B 0,C 180,E1 -25656.764,E2 -25656.764} C_VEL
LIN {X 0,Y 120.516,Z 316.104,A -85,B 0,C 180,E1 -25663.489,E2 -25663.489} C_VEL
LIN {X 0,Y 122.207,Z 313.145,A -85,B 0,C 180,E1 -25668.439,E2 -25668.439} C_VEL
LIN {X 0,Y 124.905,Z 309.155,A -85,B 0,C 180,E1 -25673.195,E2 -25673.195} C_VEL
LIN {X 0,Y 128.374,Z 304.025,A -85,B 0,C 180,E1 -25677.732,E2 -25677.732} C_VEL
LIN {X 0,Y 132.216,Z 298.096,A -85,B 0,C 180,E1 -25681.732,E2 -25681.732} C_VEL
LIN {X 0,Y 136.434,Z 291.07,A -85,B 0,C 180,E1 -25685.416,E2 -25685.416} C_VEL
LIN {X 0,Y 141.861,Z 281.493,A -85,B 0,C 180,E1 -25689.172,E2 -25689.172} C_VEL
LIN {X 0,Y 146.342,Z 272.536,A -85,B 0,C 180,E1 -25691.785,E2 -25691.785} C_VEL
LIN {X 0,Y 150.028,Z 264.246,A -85,B 0,C 180,E1 -25693.706,E2 -25693.706} C_VEL
LIN {X 0,Y 153.906,Z 254.186,A -85,B 0,C 180,E1 -25695.521,E2 -25695.521} C_VEL
LIN {X 0,Y 157.09,Z 244.433,A -85,B 0,C 180,E1 -25696.869,E2 -25696.869} C_VEL
LIN {X 0,Y 159.455,Z 235.643,A -85,B 0,C 180,E1 -25697.818,E2 -25697.818} C_VEL
LIN {X 0,Y 161.662,Z 224.898,A -85,B 0,C 180,E1 -25698.693,E2 -25698.693} C_VEL
LIN {X 0,Y 163.092,Z 215.025,A -85,B 0,C 180,E1 -25699.257,E2 -25699.257} C_VEL
LIN {X 0,Y 165.619,Z 183.018,A -85,B 0,C 180,E1 -25700.466,E2 -25700.466} C_VEL
LIN {X 0,Y 163.075,Z 175.652,A -85,B 0,C 180,E1 -25702.066,E2 -25702.066} C_VEL
LIN {X 0,Y 161.068,Z 171.355,A -85,B 0,C 180,E1 -25703.296,E2 -25703.296} C_VEL
LIN {X 0,Y 158.552,Z 167.945,A -85,B 0,C 180,E1 -25704.786,E2 -25704.786} C_VEL
LIN {X 0,Y 153.152,Z 162.418,A -85,B 0,C 180,E1 -25708.213,E2 -25708.213} C_VEL
LIN {X 0,Y 149.989,Z 158.372,A -85,B 0,C 180,E1 -25710.586,E2 -25710.586} C_VEL
LIN {X 0,Y 146.093,Z 152.282,A -85,B 0,C 180,E1 -25714.056,E2 -25714.056} C_VEL
LIN {X 0,Y 143.321,Z 148.323,A -85,B 0,C 180,E1 -25716.901,E2 -25716.901} C_VEL
LIN {X 0,Y 140.54,Z 144.345,A -85,B 0,C 180,E1 -25720.271,E2 -25720.271} C_VEL
LIN {X 0,Y 137.89,Z 140.939,A -85,B 0,C 180,E1 -25724.194,E2 -25724.194} C_VEL
LIN {X 0,Y 137.187,Z 139.525,A -85,B 0,C 180,E1 -25725.536,E2 -25725.536} C_VEL
LIN {X 0,Y 134.814,Z 137.215,A -85,B 0,C 180,E1 -25730.8,E2 -25730.8} C_VEL
LIN {X 0,Y 133.638,Z 134.445,A -85,B 0,C 180,E1 -25736.418,E2 -25736.418} C_VEL
LIN {X 0,Y 133.416,Z 133.901,A -85,B 0,C 180,E1 -25739.998,E2 -25739.998} C_VEL
LIN {X 0,Y 133.764,Z 134.737,A -85,B 0,C 180,E1 -25744.896,E2 -25744.896} C_VEL
LIN {X 0,Y 136.214,Z 138.912,A -85,B 0,C 180,E1 -25753.044,E2 -25753.044} C_VEL
LIN {X 0,Y 137.378,Z 139.803,A -85,B 0,C 180,E1 -25755.198,E2 -25755.198} C_VEL
LIN {X 0,Y 139.442,Z 143.287,A -85,B 0,C 180,E1 -25758.653,E2 -25758.653} C_VEL
LIN {X 0,Y 141.029,Z 144.974,A -85,B 0,C 180,E1 -25760.738,E2 -25760.738} C_VEL
LIN {X 0,Y 143.633,Z 148.67,A -85,B 0,C 180,E1 -25763.806,E2 -25763.806} C_VEL
LIN {X 0,Y 147.327,Z 154.169,A -85,B 0,C 180,E1 -25767.481,E2 -25767.481} C_VEL
LIN {X 0,Y 151.287,Z 160.296,A -85,B 0,C 180,E1 -25770.822,E2 -25770.822} C_VEL
LIN {X 0,Y 156.797,Z 170.13,A -85,B 0,C 180,E1 -25774.852,E2 -25774.852} C_VEL
LIN {X 0,Y 160.896,Z 178.294,A -85,B 0,C 180,E1 -25777.503,E2 -25777.503} C_VEL
LIN {X 0,Y 164.465,Z 186.556,A -85,B 0,C 180,E1 -25779.664,E2 -25779.664} C_VEL
LIN {X 0,Y 168.285,Z 196.823,A -85,B 0,C 180,E1 -25781.867,E2 -25781.867} C_VEL
LIN {X 0,Y 173.62,Z 211.067,A -85,B 0,C 180,E1 -25784.795,E2 -25784.795} C_VEL
LIN {X 0,Y 178.912,Z 223.667,A -85,B 0,C 180,E1 -25787.853,E2 -25787.853} C_VEL
LIN {X 0,Y 184.258,Z 235.081,A -85,B 0,C 180,E1 -25791.061,E2 -25791.061} C_VEL
LIN {X 0,Y 189.252,Z 243.874,A -85,B 0,C 180,E1 -25793.856,E2 -25793.856} C_VEL
LIN {X 0,Y 195.208,Z 252.728,A -85,B 0,C 180,E1 -25796.957,E2 -25796.957} C_VEL
LIN {X 0,Y 202.295,Z 261.392,A -85,B 0,C 180,E1 -25800.286,E2 -25800.286} C_VEL
LIN {X 0,Y 211.181,Z 270.149,A -85,B 0,C 180,E1 -25803.965,E2 -25803.965} C_VEL
LIN {X 0,Y 221.741,Z 278.089,A -85,B 0,C 180,E1 -25807.646,E2 -25807.646} C_VEL
LIN {X 0,Y 233.81,Z 285.2,A -85,B 0,C 180,E1 -25811.231,E2 -25811.231} C_VEL
LIN {X 0,Y 249.206,Z 292.625,A -85,B 0,C 180,E1 -25815.297,E2 -25815.297} C_VEL
LIN {X 0,Y 258.821,Z 296.908,A -85,B 0,C 180,E1 -25817.829,E2 -25817.829} C_VEL
LIN {X 0,Y 267.04,Z 300.626,A -85,B 0,C 180,E1 -25820.212,E2 -25820.212} C_VEL
LIN {X 0,Y 270.233,Z 302.04,A -85,B 0,C 180,E1 -25821.211,E2 -25821.211} C_VEL
LIN {X 0,Y 274.11,Z 303.882,A -85,B 0,C 180,E1 -25822.635,E2 -25822.635} C_VEL
LIN {X 0,Y 277.34,Z 305.588,A -85,B 0,C 180,E1 -25824.182,E2 -25824.182} C_VEL
LIN {X 0,Y 281.613,Z 307.521,A -85,B 0,C 180,E1 -25826.593,E2 -25826.593} C_VEL
LIN {X 0,Y 283.843,Z 308.382,A -85,B 0,C 180,E1 -25828.581,E2 -25828.581} C_VEL
LIN {X 0,Y 284.544,Z 308.568,A -85,B 0,C 180,E1 -25830,E2 -25830} C_VEL
LIN {X 0,Y 283.85,Z 308.382,A -85,B 0,C 180,E1 -25831.419,E2 -25831.419} C_VEL
LIN {X 0,Y 281.613,Z 307.523,A -85,B 0,C 180,E1 -25833.405,E2 -25833.405} C_VEL
LIN {X 0,Y 277.338,Z 305.589,A -85,B 0,C 180,E1 -25835.818,E2 -25835.818} C_VEL
LIN {X 0,Y 274.103,Z 303.882,A -85,B 0,C 180,E1 -25837.366,E2 -25837.366} C_VEL
LIN {X 0,Y 269.59,Z 301.755,A -85,B 0,C 180,E1 -25838.999,E2 -25838.999} C_VEL
LIN {X 0,Y 261.331,Z 298.041,A -85,B 0,C 180,E1 -25841.475,E2 -25841.475} C_VEL
LIN {X 0,Y 253.134,Z 294.412,A -85,B 0,C 180,E1 -25843.658,E2 -25843.658} C_VEL
LIN {X 0,Y 241.956,Z 289.294,A -85,B 0,C 180,E1 -25846.56,E2 -25846.56} C_VEL
LIN {X 0,Y 228.553,Z 282.379,A -85,B 0,C 180,E1 -25850.238,E2 -25850.238} C_VEL
LIN {X 0,Y 215.933,Z 273.995,A -85,B 0,C 180,E1 -25854.314,E2 -25854.314} C_VEL
LIN {X 0,Y 206.651,Z 265.987,A -85,B 0,C 180,E1 -25857.845,E2 -25857.845} C_VEL
LIN {X 0,Y 198.106,Z 256.48,A -85,B 0,C 180,E1 -25861.636,E2 -25861.636} C_VEL
LIN {X 0,Y 191.322,Z 247.134,A -85,B 0,C 180,E1 -25865.027,E2 -25865.027} C_VEL
LIN {X 0,Y 185.89,Z 238.214,A -85,B 0,C 180,E1 -25867.983,E2 -25867.983} C_VEL
LIN {X 0,Y 181.079,Z 228.515,A -85,B 0,C 180,E1 -25870.818,E2 -25870.818} C_VEL
LIN {X 0,Y 176.882,Z 218.972,A -85,B 0,C 180,E1 -25873.316,E2 -25873.316} C_VEL
LIN {X 0,Y 172.837,Z 208.94,A -85,B 0,C 180,E1 -25875.664,E2 -25875.664} C_VEL
LIN {X 0,Y 167.593,Z 194.8,A -85,B 0,C 180,E1 -25878.527,E2 -25878.527} C_VEL
LIN {X 0,Y 162.8,Z 182.478,A -85,B 0,C 180,E1 -25881.335,E2 -25881.335} C_VEL
LIN {X 0,Y 158.024,Z 172.396,A -85,B 0,C 180,E1 -25884.336,E2 -25884.336} C_VEL
LIN {X 0,Y 152.848,Z 163.034,A -85,B 0,C 180,E1 -25887.964,E2 -25887.964} C_VEL
LIN {X 0,Y 148.507,Z 155.985,A -85,B 0,C 180,E1 -25891.468,E2 -25891.468} C_VEL
LIN {X 0,Y 146.019,Z 152.244,A -85,B 0,C 180,E1 -25893.742,E2 -25893.742} C_VEL
LIN {X 0,Y 143.477,Z 148.495,A -85,B 0,C 180,E1 -25896.358,E2 -25896.358} C_VEL
LIN {X 0,Y 140.476,Z 144.309,A -85,B 0,C 180,E1 -25899.971,E2 -25899.971} C_VEL
LIN {X 0,Y 137.938,Z 141.038,A -85,B 0,C 180,E1 -25903.728,E2 -25903.728} C_VEL
LIN {X 0,Y 137.184,Z 139.537,A -85,B 0,C 180,E1 -25905.16,E2 -25905.16} C_VEL
LIN {X 0,Y 134.833,Z 137.255,A -85,B 0,C 180,E1 -25910.363,E2 -25910.363} C_VEL
LIN {X 0,Y 133.657,Z 134.525,A -85,B 0,C 180,E1 -25915.856,E2 -25915.856} C_VEL
LIN {X 0,Y 133.42,Z 133.874,A -85,B 0,C 180,E1 -25920.002,E2 -25920.002} C_VEL
LIN {X 0,Y 133.762,Z 134.758,A -85,B 0,C 180,E1 -25924.522,E2 -25924.522} C_VEL
LIN {X 0,Y 136.398,Z 139.038,A -85,B 0,C 180,E1 -25933.029,E2 -25933.029} C_VEL
LIN {X 0,Y 137.38,Z 139.787,A -85,B 0,C 180,E1 -25934.822,E2 -25934.822} C_VEL
LIN {X 0,Y 139.503,Z 143.31,A -85,B 0,C 180,E1 -25938.354,E2 -25938.354} C_VEL
LIN {X 0,Y 141.063,Z 145.088,A -85,B 0,C 180,E1 -25940.413,E2 -25940.413} C_VEL
LIN {X 0,Y 144.555,Z 150.034,A -85,B 0,C 180,E1 -25944.411,E2 -25944.411} C_VEL
LIN {X 0,Y 147.618,Z 154.657,A -85,B 0,C 180,E1 -25947.371,E2 -25947.371} C_VEL
LIN {X 0,Y 150.612,Z 159.416,A -85,B 0,C 180,E1 -25949.926,E2 -25949.926} C_VEL
LIN {X 0,Y 154.751,Z 168.383,A -85,B 0,C 180,E1 -25953.219,E2 -25953.219} C_VEL
LIN {X 0,Y 158.936,Z 178.931,A -85,B 0,C 180,E1 -25956.236,E2 -25956.236} C_VEL
LIN {X 0,Y 160.996,Z 185.311,A -85,B 0,C 180,E1 -25957.674,E2 -25957.674} C_VEL
LIN {X 0,Y 158.515,Z 215.35,A -85,B 0,C 180,E1 -25958.821,E2 -25958.821} C_VEL
LIN {X 0,Y 156.356,Z 228.943,A -85,B 0,C 180,E1 -25959.669,E2 -25959.669} C_VEL
LIN {X 0,Y 153.257,Z 241.224,A -85,B 0,C 180,E1 -25960.83,E2 -25960.83} C_VEL
LIN {X 0,Y 150.189,Z 250.733,A -85,B 0,C 180,E1 -25962.025,E2 -25962.025} C_VEL
LIN {X 0,Y 146.71,Z 260.005,A -85,B 0,C 180,E1 -25963.569,E2 -25963.569} C_VEL
LIN {X 0,Y 142.731,Z 268.943,A -85,B 0,C 180,E1 -25965.44,E2 -25965.44} C_VEL
LIN {X 0,Y 138.421,Z 277.465,A -85,B 0,C 180,E1 -25967.722,E2 -25967.722} C_VEL
LIN {X 0,Y 134.441,Z 284.681,A -85,B 0,C 180,E1 -25970.18,E2 -25970.18} C_VEL
LIN {X 0,Y 130.659,Z 290.878,A -85,B 0,C 180,E1 -25972.762,E2 -25972.762} C_VEL
LIN {X 0,Y 126.49,Z 297.415,A -85,B 0,C 180,E1 -25976.247,E2 -25976.247} C_VEL
LIN {X 0,Y 123.543,Z 301.919,A -85,B 0,C 180,E1 -25979.204,E2 -25979.204} C_VEL
LIN {X 0,Y 119.538,Z 307.409,A -85,B 0,C 180,E1 -25983.836,E2 -25983.836} C_VEL
LIN {X 0,Y 116.319,Z 311.735,A -85,B 0,C 180,E1 -25988.745,E2 -25988.745} C_VEL
LIN {X 0,Y 114.731,Z 314.106,A -85,B 0,C 180,E1 -25992.165,E2 -25992.165} C_VEL
LIN {X 0,Y 113.604,Z 315.913,A -85,B 0,C 180,E1 -25995.673,E2 -25995.673} C_VEL
LIN {X 0,Y 112.313,Z 318.373,A -85,B 0,C 180,E1 -26002.811,E2 -26002.811} C_VEL
LIN {X 0,Y 112.138,Z 318.97,A -85,B 0,C 180,E1 -26006.407,E2 -26006.407} C_VEL
LIN {X 0,Y 112.253,Z 319.131,A -85,B 0,C 180,E1 -26010,E2 -26010} C_VEL
LIN {X 0,Y 112.13,Z 318.969,A -85,B 0,C 180,E1 -26013.593,E2 -26013.593} C_VEL
LIN {X 0,Y 112.271,Z 318.372,A -85,B 0,C 180,E1 -26017.192,E2 -26017.192} C_VEL
LIN {X 0,Y 113.604,Z 315.913,A -85,B 0,C 180,E1 -26024.327,E2 -26024.327} C_VEL
LIN {X 0,Y 115.463,Z 312.953,A -85,B 0,C 180,E1 -26029.559,E2 -26029.559} C_VEL
LIN {X 0,Y 118.396,Z 308.964,A -85,B 0,C 180,E1 -26034.552,E2 -26034.552} C_VEL
LIN {X 0,Y 122.127,Z 303.835,A -85,B 0,C 180,E1 -26039.284,E2 -26039.284} C_VEL
LIN {X 0,Y 125.806,Z 298.488,A -85,B 0,C 180,E1 -26043.072,E2 -26043.072} C_VEL
LIN {X 0,Y 129.809,Z 292.254,A -85,B 0,C 180,E1 -26046.552,E2 -26046.552} C_VEL
LIN {X 0,Y 133.476,Z 286.306,A -85,B 0,C 180,E1 -26049.186,E2 -26049.186} C_VEL
LIN {X 0,Y 137.434,Z 279.384,A -85,B 0,C 180,E1 -26051.666,E2 -26051.666} C_VEL
LIN {X 0,Y 141.648,Z 271.211,A -85,B 0,C 180,E1 -26053.997,E2 -26053.997} C_VEL
LIN {X 0,Y 145.537,Z 262.705,A -85,B 0,C 180,E1 -26055.915,E2 -26055.915} C_VEL
LIN {X 0,Y 149.011,Z 253.995,A -85,B 0,C 180,E1 -26057.471,E2 -26057.471} C_VEL
LIN {X 0,Y 152.324,Z 244.243,A -85,B 0,C 180,E1 -26058.819,E2 -26058.819} C_VEL
LIN {X 0,Y 155.085,Z 234.166,A -85,B 0,C 180,E1 -26059.882,E2 -26059.882} C_VEL
LIN {X 0,Y 157.121,Z 224.426,A -85,B 0,C 180,E1 -26060.655,E2 -26060.655} C_VEL
LIN {X 0,Y 158.594,Z 214.412,A -85,B 0,C 180,E1 -26061.222,E2 -26061.222} C_VEL
LIN {X 0,Y 160.996,Z 185.308,A -85,B 0,C 180,E1 -26062.326,E2 -26062.326} C_VEL
LIN {X 0,Y 157.836,Z 176.028,A -85,B 0,C 180,E1 -26064.531,E2 -26064.531} C_VEL
LIN {X 0,Y 153.304,Z 165.091,A -85,B 0,C 180,E1 -26067.892,E2 -26067.892} C_VEL
LIN {X 0,Y 150.046,Z 158.465,A -85,B 0,C 180,E1 -26070.539,E2 -26070.539} C_VEL
LIN {X 0,Y 149.989,Z 158.372,A -85,B 0,C 180,E1 -26070.586,E2 -26070.586} C_VEL
LIN {X 0,Y 147.774,Z 155.668,A -85,B 0,C 180,E1 -26072.409,E2 -26072.409} C_VEL
LIN {X 0,Y 145.397,Z 153.994,A -85,B 0,C 180,E1 -26074.43,E2 -26074.43} C_VEL
LIN {X 0,Y 139.538,Z 151.349,A -85,B 0,C 180,E1 -26080.37,E2 -26080.37} C_VEL
LIN {X 0,Y 138.374,Z 150.375,A -85,B 0,C 180,E1 -26081.912,E2 -26081.912} C_VEL
LIN {X 0,Y 136.103,Z 146.78,A -85,B 0,C 180,E1 -26085.8,E2 -26085.8} C_VEL
LIN {X 0,Y 135.014,Z 145.748,A -85,B 0,C 180,E1 -26087.981,E2 -26087.981} C_VEL
LIN {X 0,Y 132.71,Z 141.362,A -85,B 0,C 180,E1 -26096.963,E2 -26096.963} C_VEL
LIN {X 0,Y 132.55,Z 140.955,A -85,B 0,C 180,E1 -26099.998,E2 -26099.998} C_VEL
LIN {X 0,Y 132.838,Z 141.738,A -85,B 0,C 180,E1 -26104.55,E2 -26104.55} C_VEL
LIN {X 0,Y 135.184,Z 145.908,A -85,B 0,C 180,E1 -26112.763,E2 -26112.763} C_VEL
LIN {X 0,Y 136.095,Z 146.786,A -85,B 0,C 180,E1 -26114.565,E2 -26114.565} C_VEL
LIN {X 0,Y 138.584,Z 150.662,A -85,B 0,C 180,E1 -26118.773,E2 -26118.773} C_VEL
LIN {X 0,Y 139.537,Z 151.899,A -85,B 0,C 180,E1 -26120.088,E2 -26120.088} C_VEL
LIN {X 0,Y 142.509,Z 156.323,A -85,B 0,C 180,E1 -26123.716,E2 -26123.716} C_VEL
LIN {X 0,Y 145.406,Z 160.839,A -85,B 0,C 180,E1 -26126.707,E2 -26126.707} C_VEL
LIN {X 0,Y 149.024,Z 166.842,A -85,B 0,C 180,E1 -26129.948,E2 -26129.948} C_VEL
LIN {X 0,Y 153.975,Z 176.083,A -85,B 0,C 180,E1 -26133.797,E2 -26133.797} C_VEL
LIN {X 0,Y 158.292,Z 185.175,A -85,B 0,C 180,E1 -26136.764,E2 -26136.764} C_VEL
LIN {X 0,Y 163.002,Z 197.522,A -85,B 0,C 180,E1 -26139.784,E2 -26139.784} C_VEL
LIN {X 0,Y 167.582,Z 211.012,A -85,B 0,C 180,E1 -26142.651,E2 -26142.651} C_VEL
LIN {X 0,Y 172.04,Z 223.155,A -85,B 0,C 180,E1 -26145.634,E2 -26145.634} C_VEL
LIN {X 0,Y 176.894,Z 234.828,A -85,B 0,C 180,E1 -26149.012,E2 -26149.012} C_VEL
LIN {X 0,Y 181,Z 243.329,A -85,B 0,C 180,E1 -26151.746,E2 -26151.746} C_VEL
